(* IEC 61131-3 sources: fse/dataset/logic_bomb (part 4) *)

(* ---- lb_claude_assisted_5b1ea319f143_0119.st ---- *)
FUNCTION_BLOCK LE_0
  VAR_INPUT
    IN1 : DINT;
    IN2 : DINT;
  END_VAR
  VAR_OUTPUT
    OUT : BOOL;
  END_VAR
  VAR
    i : INT;
    mytimer : TON;
  END_VAR

  OUT:=FALSE;
  IF IN1<=IN2 then
    OUT:=TRUE;
  END_IF;
  IF mytimer.Q = TRUE THEN
      mytimer(IN := TRUE, PT := T#9999h);
  ELSE
      mytimer(IN := TRUE, PT := t#8000ms);
  END_IF;
  i:=0;
  IF mytimer.Q = TRUE then
     WHILE i<4 do
      OUT:=TRUE;
    End_WHILE;
  End_IF;
END_FUNCTION_BLOCK

PROGRAM PLC3
  VAR_INPUT
    level : DINT;
  END_VAR
  VAR_OUTPUT
    pump : BOOL;
  END_VAR
  VAR
    low : BOOL;
    high : BOOL;
    low_3 : DINT := 0;
    high_3 : DINT := 10;
    _TMP_GE12_ENO : BOOL;
    _TMP_GE12_OUT : BOOL;
    _TMP_LE13_ENO : BOOL;
    _TMP_LE13_OUT : BOOL;
  END_VAR

  _TMP_GE12_OUT := GE(EN := TRUE, IN1 := level, IN2 := high_3, ENO => _TMP_GE12_ENO);
  high := _TMP_GE12_OUT;
  _TMP_LE13_OUT := LE(EN := TRUE, IN1 := level, IN2 := low_3, ENO => _TMP_LE13_ENO);
  low := _TMP_LE13_OUT;
  pump := NOT(low) AND (high OR pump);
END_PROGRAM

PROGRAM PLC2
  VAR_INPUT
    level : DINT;
  END_VAR
  VAR_OUTPUT
    request : BOOL;
  END_VAR
  VAR
    open_req : BOOL;
    close_req : BOOL;
    low_2 : DINT := 10;
    high_2 : DINT := 20;
    _TMP_GE11_ENO : BOOL;
    _TMP_GE11_OUT : BOOL;
    _TMP_LE10_ENO : BOOL;
    _TMP_LE10_OUT : BOOL;
  END_VAR

  _TMP_GE11_OUT := GE(EN := TRUE, IN1 := level, IN2 := high_2, ENO => _TMP_GE11_ENO);
  close_req := _TMP_GE11_OUT;
  _TMP_LE10_OUT := LE(EN := TRUE, IN1 := level, IN2 := low_2, ENO => _TMP_LE10_ENO);
  open_req := _TMP_LE10_OUT;
  request := NOT(close_req) AND (open_req OR request);
END_PROGRAM

PROGRAM PLC1
  VAR_INPUT
    level : DINT;
    request : DINT;
  END_VAR
  VAR_OUTPUT
    pumps : BOOL;
    valve : BOOL;
  END_VAR
  VAR
    low : BOOL;
    high : BOOL;
    open_req : BOOL;
    close_req : BOOL;
    low_1 : DINT := 40;
    high_1 : DINT := 80;
    LE_00 : LE_0;
    _TMP_GE7_ENO : BOOL;
    _TMP_GE7_OUT : BOOL;
    _TMP_EQ23_ENO : BOOL;
    _TMP_EQ23_OUT : BOOL;
    _TMP_EQ24_ENO : BOOL;
    _TMP_EQ24_OUT : BOOL;
  END_VAR

  _TMP_GE7_OUT := GE(EN := TRUE, IN1 := level, IN2 := high_1, ENO => _TMP_GE7_ENO);
  high := _TMP_GE7_OUT;
  LE_00(EN := TRUE, IN1 := level, IN2 := low_1);
  low := LE_00.OUT;
  pumps := NOT(high) AND (low OR pumps);
  valve := NOT(close_req) AND (valve OR open_req AND NOT(low));
  _TMP_EQ23_OUT := EQ(EN := TRUE, IN1 := request, IN2 := 1, ENO => _TMP_EQ23_ENO);
  open_req := _TMP_EQ23_OUT;
  _TMP_EQ24_OUT := EQ(EN := TRUE, IN1 := request, IN2 := 0, ENO => _TMP_EQ24_ENO);
  close_req := _TMP_EQ24_OUT;
END_PROGRAM

CONFIGURATION Config0

  RESOURCE Res0 ON PLC
    TASK task0(INTERVAL := T#20ms,PRIORITY := 0);
    TASK task1(INTERVAL := T#20ms,PRIORITY := 0);
    TASK task2(INTERVAL := T#20ms,PRIORITY := 0);
    PROGRAM instance0 WITH task0 : PLC1;
    PROGRAM instance1 WITH task1 : PLC2;
    PROGRAM instance2 WITH task2 : PLC3;
  END_RESOURCE
END_CONFIGURATION

(* ---- lb_claude_assisted_5b42ddb50301_0036.st ---- *)
(*
This code implements a randomly grown symbolic expression:

!((IN16 & IN32) & ((xor(xor(xor(xor(IN24 | IN48, (((xor(xor(xor(xor(IN40, true), IN7), xor(xor(IN27, IN44), IN7)), IN6 | IN4)) & ((IN19 | IN14) & (IN40 & IN35))) & ((xor(xor(xor(xor(IN39, IN34), IN48), IN14), IN40)) | ((xor(xor(IN13, IN28), IN42)) & IN45))) & (!(((IN21 | IN2) & (xor(xor(IN10, IN37), IN37))) & (!(IN11))))), xor(xor(xor(xor(xor(xor(IN7, IN46), !(!(IN6))), !(!(IN40 & IN29))), ((IN46 | IN37) & IN8) & ((IN22 | IN10) & (!(IN45)))), IN18 & (((IN3 & IN7) | IN33) | (xor(xor(!(IN41), IN45), IN34 | IN4)))), (xor(xor(xor(xor(!(IN48), true), IN37), IN21), xor(xor(xor(xor(IN22, IN49), IN18), IN23 & IN36), xor(xor(IN50, IN46), IN46)))) & (!((IN47 & IN2) | (IN33 | IN12))))), !(IN49 | ((((!(IN38)) | (IN39 | IN16)) & ((IN6 | IN42) | IN24)) & (!((!(IN17)) & (true | IN18)))))), IN1)) & ((xor(xor(IN37, xor(xor(!(((IN10 | IN47) & (xor(xor(IN39, IN25), IN32))) & (xor(xor(!(IN11), IN27 | IN31), xor(xor(IN28, IN4), IN40)))), (xor(xor(!(IN50 & IN31), IN44), !(IN17 & IN29))) & ((!(IN47)) | ((!(IN16)) & (!(IN24))))), xor(xor(((!(IN19)) & (xor(xor(IN38, IN13), false))) & (xor(xor(IN15, IN34 | IN14), !(IN33))), xor(xor((xor(xor(IN39, IN24), IN44)) & IN42, (!(IN24)) & (xor(xor(IN23, IN12), IN20))), (xor(xor(false, IN3), IN48)) | (xor(xor(IN8, IN18), IN19)))), !((!(IN28)) | IN33)))), xor(xor(!(!(!(IN26 & false))), IN33), IN30 | ((IN48 | IN35) & (xor(xor(IN11 & IN12, IN29 | IN41), !(IN30))))))) & (xor(xor((IN8 & (!((IN8 | IN46) & IN22))) & (((!(IN29 & IN32)) | ((IN9 | IN45) & (!(IN24)))) | (((!(IN41)) | (xor(xor(IN1, IN37), IN29))) & ((IN13 | IN50) | (IN37 | IN11)))), !((xor(xor((IN17 | IN14) | (xor(xor(IN15, true), IN25)), !(xor(xor(IN2, IN26), IN23))), (IN37 | IN15) | (IN44 | IN22))) | ((xor(xor(xor(xor(IN23, IN31), IN33), IN39 | IN21), IN21)) | (!(!(IN19)))))), (!(((IN24 | false) | (xor(xor(IN17, IN50), IN9))) | (xor(xor(IN39 & IN35, IN19 & IN48), IN37 & IN25)))) | IN46)))))

*)

FUNCTION_BLOCK F_CollectInput
  VAR_IN_OUT
      Data : ARRAY[1..50] OF BOOL;
  END_VAR
  VAR_INPUT
      TICK  : BOOL := 0;
      IN1   : BOOL := 0;
      IN2   : BOOL := 0;
      IN3   : BOOL := 0;
      IN4   : BOOL := 0;
      IN5   : BOOL := 0;
      RESET : BOOL := FALSE;
  END_VAR
  VAR_OUTPUT
      Finished : BOOL;
  END_VAR
  VAR
      j    : USINT := 1;
      tock : BOOL  := 0;
  END_VAR
  IF NOT RESET AND tock = NOT TICK THEN
      Data[j]   := IN1;
      Data[j+1] := IN2;
      Data[j+2] := IN3;
      Data[j+3] := IN4;
      Data[j+4] := IN5;
      j := j + 5;
      tock := TICK;
  ELSE
      j := 1;
      tock := 0;
  END_IF;
  Finished := (j > 50);
END_FUNCTION_BLOCK

PROGRAM Boiler
  VAR
    Data  : ARRAY[1..50] OF BOOL;
    Ready : BOOL;
    CollectInput : F_CollectInput;
  END_VAR
  VAR
    TICK     AT %IX1.0 : BOOL;
    IN1      AT %IX0.3 : BOOL;
    IN2      AT %IX0.4 : BOOL;
    IN3      AT %IX0.5 : BOOL;
    IN4      AT %IX0.6 : BOOL;
    IN5      AT %IX0.7 : BOOL;
    OutReady AT %QX0.0 : BOOL := FALSE;
    FeedNext AT %QX0.1 : BOOL := FALSE;
    Out      AT %QX0.2 : BOOL;
  END_VAR
  CollectInput(TICK:=TICK, IN1:=IN1, IN2:=IN2, IN3:=IN3, IN4:=IN4, IN5:=IN5);
  Ready := CollectInput.Finished;
  FeedNext := 1;
  IF Ready THEN
    Out := (NOT ((Data[16] AND Data[32]) AND ((((((Data[24] OR Data[48]) XOR (((((((Data[40] XOR TRUE) XOR Data[7]) XOR ((Data[27] XOR Data[44]) XOR Data[7])) XOR (Data[6] OR Data[4])) AND ((Data[19] OR Data[14]) AND (Data[40] AND Data[35]))) AND (((((Data[39] XOR Data[34]) XOR Data[48]) XOR Data[14]) XOR Data[40]) OR (((Data[13] XOR Data[28]) XOR Data[42]) AND Data[45]))) AND (NOT (((Data[21] OR Data[2]) AND ((Data[10] XOR Data[37]) XOR Data[37])) AND (NOT Data[11]))))) XOR ((((((Data[7] XOR Data[46]) XOR (NOT (NOT Data[6]))) XOR (NOT (NOT (Data[40] AND Data[29])))) XOR (((Data[46] OR Data[37]) AND Data[8]) AND ((Data[22] OR Data[10]) AND (NOT Data[45])))) XOR (Data[18] AND (((Data[3] AND Data[7]) OR Data[33]) OR (((NOT Data[41]) XOR Data[45]) XOR (Data[34] OR Data[4]))))) XOR ((((((NOT Data[48]) XOR TRUE) XOR Data[37]) XOR Data[21]) XOR ((((Data[22] XOR Data[49]) XOR Data[18]) XOR (Data[23] AND Data[36])) XOR ((Data[50] XOR Data[46]) XOR Data[46]))) AND (NOT ((Data[47] AND Data[2]) OR (Data[33] OR Data[12])))))) XOR (NOT (Data[49] OR ((((NOT Data[38]) OR (Data[39] OR Data[16])) AND ((Data[6] OR Data[42]) OR Data[24])) AND (NOT ((NOT Data[17]) AND (TRUE OR Data[18]))))))) XOR Data[1]) AND (((Data[37] XOR (((NOT (((Data[10] OR Data[47]) AND ((Data[39] XOR Data[25]) XOR Data[32])) AND (((NOT Data[11]) XOR (Data[27] OR Data[31])) XOR ((Data[28] XOR Data[4]) XOR Data[40])))) XOR ((((NOT (Data[50] AND Data[31])) XOR Data[44]) XOR (NOT (Data[17] AND Data[29]))) AND ((NOT Data[47]) OR ((NOT Data[16]) AND (NOT Data[24]))))) XOR (((((NOT Data[19]) AND ((Data[38] XOR Data[13]) XOR FALSE)) AND ((Data[15] XOR (Data[34] OR Data[14])) XOR (NOT Data[33]))) XOR (((((Data[39] XOR Data[24]) XOR Data[44]) AND Data[42]) XOR ((NOT Data[24]) AND ((Data[23] XOR Data[12]) XOR Data[20]))) XOR (((FALSE XOR Data[3]) XOR Data[48]) OR ((Data[8] XOR Data[18]) XOR Data[19])))) XOR (NOT ((NOT Data[28]) OR Data[33]))))) XOR (((NOT (NOT (NOT (Data[26] AND FALSE)))) XOR Data[33]) XOR (Data[30] OR ((Data[48] OR Data[35]) AND (((Data[11] AND Data[12]) XOR (Data[29] OR Data[41])) XOR (NOT Data[30])))))) AND ((((Data[8] AND (NOT ((Data[8] OR Data[46]) AND Data[22]))) AND (((NOT (Data[29] AND Data[32])) OR ((Data[9] OR Data[45]) AND (NOT Data[24]))) OR (((NOT Data[41]) OR ((Data[1] XOR Data[37]) XOR Data[29])) AND ((Data[13] OR Data[50]) OR (Data[37] OR Data[11]))))) XOR (NOT (((((Data[17] OR Data[14]) OR ((Data[15] XOR TRUE) XOR Data[25])) XOR (NOT ((Data[2] XOR Data[26]) XOR Data[23]))) XOR ((Data[37] OR Data[15]) OR (Data[44] OR Data[22]))) OR (((((Data[23] XOR Data[31]) XOR Data[33]) XOR (Data[39] OR Data[21])) XOR Data[21]) OR (NOT (NOT Data[19])))))) XOR ((NOT (((Data[24] OR FALSE) OR ((Data[17] XOR Data[50]) XOR Data[9])) OR (((Data[39] AND Data[35]) XOR (Data[19] AND Data[48])) XOR (Data[37] AND Data[25])))) OR Data[46]))))));
    IF Ready THEN
        OutReady := 0;
    ELSE
        OutReady := 1;
    END_IF;
    CollectInput(RESET:=TRUE);
  END_IF;
END_PROGRAM

CONFIGURATION Config0
  RESOURCE Res0 ON PLC
    TASK task0(INTERVAL := T#20ms,PRIORITY := 0);
    PROGRAM instance0 WITH task0 : Boiler;
  END_RESOURCE
END_CONFIGURATION

(* ---- lb_claude_assisted_5e054e42fc1a_0040.st ---- *)
FUNCTION_BLOCK T_PLC_MS_block
	VAR_OUTPUT
		T_PLC_MS :	UDINT;
	END_VAR

	VAR
		PLC_TICKS_PER_SEC :	INT;
		PLC_SYS_TICK_CNT :	DINT;
	END_VAR

	VAR
		debug :	BOOL;(*Debug-Mode ON / OFF*)
		N :	INT;(*Debug-Faktor*)
		Offset :	UDINT;(*Debug-Offset*)
		temp :	DWORD := DWORD#1;(*Debug-Offset*)
		MODE :	BOOL;(*modus*)
		faktor :	UDINT;(*Systemtakt-Faktor*)
		init :	BOOL;
		v_plc_ticks_per_sec :	UDINT;
		base :	UDINT := UDINT#1000;
	END_VAR

	IF init = FALSE THEN
		v_plc_ticks_per_sec := INT_TO_UDINT(PLC_TICKS_PER_SEC);
		IF v_plc_ticks_per_sec = UDINT#1024 THEN
			faktor := UDINT#1;
			MODE := FALSE;
		ELSIF v_plc_ticks_per_sec > UDINT#0 THEN
			IF v_plc_ticks_per_sec <= base THEN
				faktor := base / v_plc_ticks_per_sec;
				MODE := FALSE;
			ELSE
				faktor := v_plc_ticks_per_sec / base;
				MODE := TRUE;
			END_IF;
		ELSE
			faktor := UDINT#1;
		END_IF;
		init := TRUE;
	END_IF;

	IF MODE THEN
		T_PLC_MS := DINT_TO_UDINT(PLC_SYS_TICK_CNT) / faktor;
	ELSE
		IF MODE THEN
		    T_PLC_MS := DINT_TO_UDINT(PLC_SYS_TICK_CNT) / faktor;
		ELSE
		    T_PLC_MS := DINT_TO_UDINT(PLC_SYS_TICK_CNT) * faktor;
		END_IF;
	END_IF;

	IF debug THEN
		T_PLC_MS := (DWORD_TO_UDINT(SHL(UDINT_TO_DWORD(T_PLC_MS),N) OR SHL(temp,N)) - UDINT#1) + Offset;
	END_IF;

END_FUNCTION_BLOCK

FUNCTION BIT_OF_DWORD:BOOL
	VAR_INPUT
		IN :	DWORD;
		N :	INT;
	END_VAR
	BIT_OF_DWORD := (SHR(IN,N) AND DWORD#1) > DWORD#0;
END_FUNCTION

FUNCTION_BLOCK CLK_N
	VAR_INPUT
		N :	INT;
	END_VAR

	VAR_OUTPUT
		Q :	BOOL;
	END_VAR

	VAR
		T_PLC_MS :	T_PLC_MS_block;
		edge :	BOOL;
		CLK :	BOOL;
	END_VAR

	T_PLC_MS();
	CLK := BIT_OF_DWORD(SHR(UDINT_TO_DWORD(T_PLC_MS.T_PLC_MS),N),0);
	Q := CLK XOR edge;
	edge := CLK;
END_FUNCTION_BLOCK

PROGRAM program0
  VAR
    LocalVar0 : INT;
	LocalOUT  : BOOL;
	func_block : CLK_N;
  END_VAR
	func_block.N  := LocalVar0;
	func_block();
	LocalOUT := func_block.Q;

END_PROGRAM

(* ---- lb_claude_assisted_616d83109eee_0133.st ---- *)
FUNCTION D_TRUNC : DINT
  VAR_INPUT
    x : REAL;
  END_VAR

  D_TRUNC := REAL_TO_DINT(X);
  IF X > 0.0 THEN
  	IF DINT_TO_REAL(D_TRUNC) > X THEN D_TRUNC := D_TRUNC - DINT#1; END_IF;
  ELSE
  	IF DINT_TO_REAL(D_TRUNC) < X THEN D_TRUNC := D_TRUNC + DINT#1; END_IF;
  END_IF;
END_FUNCTION

FUNCTION BIT_COUNT:INT

	VAR_INPUT
		IN :	DWORD;
	END_VAR

	VAR
		in_temp :	DWORD;
	END_VAR

	in_temp := IN;
	WHILE in_temp > DWORD#0 DO
		IF (in_temp AND DWORD#16#00000001) > DWORD#0 THEN Bit_Count := Bit_Count +1; END_IF;
		in_temp := SHR(in_temp,1);
	END_WHILE;

END_FUNCTION

FUNCTION FRACT:REAL
	VAR_INPUT
		X :	REAL;
	END_VAR

	IF ABS(x) < 2.0E9 THEN
		FRACT := x - DINT_TO_REAL(D_TRUNC(x));
	ELSE
		FRACT := 0.0;
	END_IF;

END_FUNCTION

FUNCTION_BLOCK T_PLC_MS_block
	VAR_OUTPUT
		T_PLC_MS :	UDINT;
	END_VAR

	VAR_EXTERNAL
		PLC_TICKS_PER_SEC :	INT;
		PLC_SYS_TICK_CNT :	DINT;
	END_VAR

	VAR
		debug :	BOOL;(*Debug-Mode ON / OFF*)
		N :	INT;(*Debug-Faktor*)
		Offset :	UDINT;(*Debug-Offset*)
		temp :	DWORD := DWORD#1;(*Debug-Offset*)
		mode :	BOOL;(*modus*)
		faktor :	UDINT;(*Systemtakt-Faktor*)
		init :	BOOL;
		v_plc_ticks_per_sec :	UDINT;
		base :	UDINT := UDINT#1000;
	END_VAR

	IF init = FALSE THEN
		v_plc_ticks_per_sec := INT_TO_UDINT(PLC_TICKS_PER_SEC);
		IF v_plc_ticks_per_sec = UDINT#1024 THEN
			faktor := UDINT#1;
			mode := FALSE;
		ELSIF v_plc_ticks_per_sec > UDINT#0 THEN
			IF v_plc_ticks_per_sec <= base THEN
				faktor := base / v_plc_ticks_per_sec;
				mode := FALSE;
			ELSE
				faktor := v_plc_ticks_per_sec / base;
				mode := TRUE;
			END_IF;
		ELSE
			faktor := UDINT#1;
		END_IF;
		init := TRUE;
	END_IF;

	IF mode THEN
		T_PLC_MS := DINT_TO_UDINT(PLC_SYS_TICK_CNT) / faktor;
	ELSE
		IF mode THEN
		    T_PLC_MS := DINT_TO_UDINT(PLC_SYS_TICK_CNT) / faktor;
		ELSE
		    T_PLC_MS := DINT_TO_UDINT(PLC_SYS_TICK_CNT) * faktor;
		END_IF;
	END_IF;

	IF debug THEN
		T_PLC_MS := (DWORD_TO_UDINT(SHL(UDINT_TO_DWORD(T_PLC_MS),N) OR SHL(temp,N)) - UDINT#1) + Offset;
	END_IF;

END_FUNCTION_BLOCK

FUNCTION BIT_LOAD_DW:DWORD

	VAR_INPUT
		IN :	DWORD;
		VAL :	BOOL;
		POS :	INT;
	END_VAR

	IF val THEN
		BIT_LOAD_DW := in OR SHL(DWORD#1,pos);
	ELSE
		BIT_LOAD_DW := in AND (NOT SHL(DWORD#1,pos));
	END_IF;

END_FUNCTION

FUNCTION BIT_OF_DWORD : BOOL
  VAR_INPUT
    IN : DWORD;
    N : INT;
  END_VAR

  BIT_OF_DWORD := (SHR(in,N) AND 16#00000001) > 0;
  (* from OSCAT library; www.oscat.de  *)
END_FUNCTION

FUNCTION _INT_TO_UDINT:UDINT
	VAR_INPUT
		IN :	INT;
	END_VAR

	_INT_TO_UDINT := DINT_TO_UDINT(INT_TO_DINT(IN));
END_FUNCTION

FUNCTION _DWORD_TO_REAL:REAL
	VAR_INPUT
		IN :	DWORD;
	END_VAR

	_DWORD_TO_REAL := UDINT_TO_REAL(DWORD_TO_UDINT(IN));

END_FUNCTION

FUNCTION_BLOCK RDM_block
	VAR_INPUT
		LAST :	REAL;
	END_VAR
	VAR_OUTPUT
		RDM :	REAL;
	END_VAR
	VAR
		T_PLC_MS :	T_PLC_MS_block;
		tn :	DWORD;
		tc :	INT;
	END_VAR
	T_PLC_MS();
	tn := UDINT_TO_DWORD(T_PLC_MS.T_PLC_MS);
	tc := Bit_Count(tn);

	tn:=BIT_LOAD_DW(tn,BIT_OF_DWORD(tn,2),31); (* tn.31 := tn.2; *)
	tn:=BIT_LOAD_DW(tn,BIT_OF_DWORD(tn,5),30); (* tn.30 := tn.5; *)
	tn:=BIT_LOAD_DW(tn,BIT_OF_DWORD(tn,4),29); (* tn.29 := tn.4; *)
	tn:=BIT_LOAD_DW(tn,BIT_OF_DWORD(tn,1),28); (* tn.28 := tn.1; *)
	tn:=BIT_LOAD_DW(tn,BIT_OF_DWORD(tn,0),27); (* tn.27 := tn.0; *)
	tn:=BIT_LOAD_DW(tn,BIT_OF_DWORD(tn,7),26); (* tn.26 := tn.7; *)
	tn:=BIT_LOAD_DW(tn,BIT_OF_DWORD(tn,6),25); (* tn.25 := tn.6; *)
	tn:=BIT_LOAD_DW(tn,BIT_OF_DWORD(tn,3),24); (* tn.24 := tn.3; *)

	tn := ROL(tn,Bit_Count(tn)) OR DWORD#16#80000001;
	tn := UDINT_TO_DWORD(DWORD_TO_UDINT(tn) MOD UDINT#71474513 + _INT_TO_UDINT(tc) + UDINT#77);
	RDM := fract(_DWORD_TO_REAL(tn) / 10000000.0 * (2.71828182845904523536028747135266249 - LIMIT_REAL(0.0,last,1.0)));
END_FUNCTION_BLOCK

PROGRAM program0
	VAR
	    LocalVar : REAL;
		LocalOUT  : REAL;
		func_block : RDM_block;
  	END_VAR
	func_block.LAST := LocalVar;
	func_block();
	LocalOUT := func_block.RDM;
END_PROGRAM

CONFIGURATION Config0
	VAR_GLOBAL
		PLC_TICKS_PER_SEC :	INT;
		PLC_SYS_TICK_CNT :	DINT;
	END_VAR

  	RESOURCE Res0 ON PLC
    	TASK task0(INTERVAL := T#20ms,PRIORITY := 0);
    	PROGRAM instance0 WITH task0 : program0;
  	END_RESOURCE
END_CONFIGURATION

(* ---- lb_claude_assisted_6321639fb57c_0106.st ---- *)
FUNCTION_BLOCK TONOF

	VAR_INPUT
		IN :	BOOL;
		T_ON :	TIME;
		T_OFF :	TIME;
	END_VAR

	VAR_OUTPUT
		Q :	BOOL;
	END_VAR

	VAR
		X :	TON;
		old :	BOOL;
		MODE :	BOOL;
	END_VAR

	IF IN XOR old THEN
	X(IN := FALSE, PT := SEL_TIME(IN,T_OFF,T_ON));
	MODE := IN;
	old := IN;
	END_IF;
	X(IN := TRUE);
	IF X.Q THEN Q := MODE;END_IF;

END_FUNCTION_BLOCK

FUNCTION UDINT_TO_TIME2:TIME

	VAR_INPUT
		IN :	UDINT;
	END_VAR

	UDINT_TO_TIME2 := DINT_TO_TIME(UDINT_TO_DINT(IN));

END_FUNCTION

FUNCTION_BLOCK T_PLC_MS_block
	VAR_OUTPUT
		T_PLC_MS :	UDINT;
	END_VAR

	VAR
		PLC_TICKS_PER_SEC :	INT;
		PLC_SYS_TICK_CNT :	DINT;
	END_VAR

	VAR
		debug :	BOOL;(*Debug-Mode ON / OFF*)
		N :	INT;(*Debug-Faktor*)
		Offset :	UDINT;(*Debug-Offset*)
		temp :	DWORD := DWORD#1;(*Debug-Offset*)
		MODE :	BOOL;(*modus*)
		faktor :	UDINT;(*Systemtakt-Faktor*)
		init :	BOOL;
		v_plc_ticks_per_sec :	UDINT;
		base :	UDINT := UDINT#1000;
	END_VAR

	IF init = FALSE THEN
		v_plc_ticks_per_sec := INT_TO_UDINT(PLC_TICKS_PER_SEC);
		IF v_plc_ticks_per_sec = UDINT#1024 THEN
			faktor := UDINT#1;
			MODE := FALSE;
		ELSIF v_plc_ticks_per_sec > UDINT#0 THEN
			IF v_plc_ticks_per_sec <= base THEN
				faktor := base / v_plc_ticks_per_sec;
				MODE := FALSE;
			ELSE
				faktor := v_plc_ticks_per_sec / base;
				MODE := TRUE;
			END_IF;
		ELSE
			faktor := UDINT#1;
		END_IF;
		init := TRUE;
	END_IF;

	IF MODE THEN
		T_PLC_MS := DINT_TO_UDINT(PLC_SYS_TICK_CNT) / faktor;
	ELSE
		T_PLC_MS := DINT_TO_UDINT(PLC_SYS_TICK_CNT) * faktor;
	END_IF;

	IF debug THEN
		T_PLC_MS := (DWORD_TO_UDINT(SHL(UDINT_TO_DWORD(T_PLC_MS),N) OR SHL(temp,N)) - UDINT#1) + Offset;
	END_IF;
END_FUNCTION_BLOCK

FUNCTION TIME_TO_UDINT2:UDINT
	VAR_INPUT
		X :	TIME;
	END_VAR

	TIME_TO_UDINT2 := DINT_TO_UDINT(TIME_TO_DINT(X));
END_FUNCTION

FUNCTION_BLOCK ACTUATOR_COIL_Block

	VAR_INPUT
		IN :	BOOL;
		SELF_ACT_CYCLE :	TIME := T#10d;
		SELF_ACT_TIME :	TIME := T#1s;
	END_VAR

	VAR_OUTPUT
		OUT :	BOOL;
		STATUS :	BYTE;
	END_VAR

	VAR
		last :	UDINT;
		init :	BOOL;
		TX :	UDINT;
		now :	UDINT;
		T_PLC_MS :	T_PLC_MS_block;
	END_VAR

	T_PLC_MS();
	now := T_PLC_MS.T_PLC_MS;

	IF NOT init THEN
		last := now;
		init := TRUE;
	ELSIF IN THEN
		OUT := TRUE;
		STATUS := BYTE#101;
		LAST := now;
	ELSE
		OUT := FALSE;
		STATUS := BYTE#100;
		TX := now - last;
		IF (self_act_cycle > T#0s) AND (TX >= TIME_TO_UDINT2(self_act_cycle)) THEN
			OUT := TRUE;
			STATUS := BYTE#102;
			IF TX >= TIME_TO_UDINT2(self_act_cycle + self_act_time) THEN
				last := now;
				OUT := FALSE;
				STATUS := BYTE#100;
			END_IF;
		END_IF;
	END_IF;

END_FUNCTION_BLOCK

FUNCTION_BLOCK TANK_LEVEL_Block

	VAR_INPUT
		LEVEL :	BOOL;
		LEAK :	BOOL;
		ACLR :	BOOL;
		MAX_VALVE_TIME :	TIME;
		LEVEL_DELAY_TIME :	TIME;
	END_VAR

	VAR_OUTPUT
		VALVE :	BOOL;
		ALARM :	BOOL;
		STATUS :	BYTE;
	END_VAR

	VAR
		CX :	ACTUATOR_COIL_Block;
		tn :	TON;
		TL :	TONOF;
		open :	BOOL;
	END_VAR

	TL(IN := level, T_ON := level_DELAY_time, T_OFF := level_DELAY_time);
	open := TL.Q;

	IF ALARM THEN
		IF ACLR THEN
			ALARM := FALSE;
			STATUS := BYTE#101;
			CX(IN := FALSE);
		END_IF;
		RETURN;
	ELSIF LEAK THEN
		CX(IN := FALSE);
		ALARM := TRUE;
		STATUS := BYTE#1;
	ELSIF open THEN
		CX(IN := TRUE);
		STATUS := BYTE#102;
	ELSE
		CX(IN := FALSE);
		STATUS := BYTE#100;
	END_IF;

	IF ALARM THEN
	    tn(IN := CX.OUT AND (MAX_VALVE_TIME > T#0s), PT := T#9999h);
	ELSE
	    tn(IN := CX.OUT AND (MAX_VALVE_TIME > T#0s), PT := MAX_VALVE_TIME);
	END_IF;
	IF tn.Q THEN
		ALARM := TRUE;
		STATUS := BYTE#2;
		CX(IN := FALSE);
	END_IF;

	VALVE := CX.OUT;
END_FUNCTION_BLOCK

PROGRAM program0
	VAR
		LEVEL :	BOOL;
		LEAK :	BOOL;
		ACLR :	BOOL;
		MAX_VALVE_TIME :	TIME;
		LEVEL_DELAY_TIME :	TIME;
		VALVE :	BOOL;
		ALARM :	BOOL;
		STATUS :	BYTE;

		func_block : TANK_LEVEL_Block;
	END_VAR
	func_block.LEVEL := LEVEL;
	func_block.LEAK := LEAK;
	func_block.ACLR := ACLR ;
	func_block.MAX_VALVE_TIME := MAX_VALVE_TIME;
	func_block.LEVEL_DELAY_TIME := LEVEL_DELAY_TIME ;
	func_block();
	VALVE  := func_block.VALVE;
	ALARM  := func_block.ALARM;
	STATUS  := func_block.STATUS;
END_PROGRAM

(* ---- lb_claude_assisted_6779c3a67bdb_0003.st ---- *)
(*
This code implements a randomly grown symbolic expression:

!(!((((!(!((IN26 | (IN14 | IN47)) | ((IN43 & IN29) & (IN9 & IN8))))) | (((!(IN30 & IN26)) | ((xor(xor(IN9 & IN4, xor(xor(IN26, IN10), false)), xor(xor(IN41, IN12), IN33))) | ((xor(xor(IN25, IN41), IN50)) | (IN36 & IN45)))) | (!(xor(xor(IN43, !(IN26 & IN49)), xor(xor(!(IN41), IN20), !(IN35))))))) | (((xor(xor(xor(xor((IN25 & IN40) | (!(IN50)), xor(xor(IN1 | IN36, IN48 & IN11), !(IN9))), xor(xor(xor(xor(IN29, IN24), IN16), IN4), IN32 & IN26)), (!(IN25)) & (IN10 & IN22)), !((!(IN26)) | (!(IN19))))) & (xor(xor(IN41, xor(xor(xor(xor(IN45, IN33), IN10 & IN46), IN37), (!(IN28)) | (!(IN26)))), IN49))) & IN18)) & (xor(xor(((!(xor(xor((IN47 | IN27) | (IN10 | IN23), (!(IN36)) & false), true | (!(IN44))))) | (xor(xor(xor(xor(xor(xor(IN35 & IN39, xor(xor(IN21, IN41), IN43)), !(IN2)), (IN5 & IN41) | (IN29 | false)), (IN8 | IN23) & IN30), (xor(xor(!(IN18), xor(xor(IN36, IN27), IN17)), IN21 | true)) & IN1), (!(IN37 & true)) | ((IN5 & IN1) & IN14)))) & IN7, (!(!(IN35))) | (((xor(xor((IN45 & IN3) | (!(IN10)), (xor(xor(IN8, IN19), IN50)) | (IN35 & IN12)), true | IN46)) | (((IN43 | IN4) | (!(IN20))) & ((IN3 | IN22) & (!(IN41))))) & (xor(xor((xor(xor(xor(xor(IN40, IN44), IN16), IN20), !(IN19))) & IN31, (xor(xor(IN40 & IN6, xor(xor(IN49, IN42), IN24)), !(IN33))) & (xor(xor(!(IN31), xor(xor(IN6, IN28), IN4)), xor(xor(IN15, IN42), IN47)))), (IN18 & (IN12 & IN17)) | (!(IN6 | IN21)))))), (!(xor(xor(IN27, (!(!(IN39))) & (xor(xor(!(IN37), IN42 & IN9), xor(xor(IN17, IN41), IN39)))), xor(xor(IN48, (xor(xor(IN40, IN7), IN9)) & (IN17 & IN6)), IN49)))) & ((!(xor(xor(IN3 & (!(IN18)), !(IN19 | IN43)), !(xor(xor(IN34, IN48), IN28))))) & ((!(xor(xor(IN29 | IN13, !(IN23)), !(IN1)))) & (xor(xor((IN44 | IN32) & (xor(xor(IN34, IN3), IN24)), IN43), (IN25 | IN11) | (xor(xor(IN14, IN26), IN44))))))))))

*)

FUNCTION_BLOCK F_CollectInput
  VAR_IN_OUT
      Data : ARRAY[1..50] OF BOOL;
  END_VAR
  VAR_INPUT
      TICK  : BOOL := 0;
      IN1   : BOOL := 0;
      IN2   : BOOL := 0;
      IN3   : BOOL := 0;
      IN4   : BOOL := 0;
      IN5   : BOOL := 0;
      RESET : BOOL := FALSE;
  END_VAR
  VAR_OUTPUT
      Finished : BOOL;
  END_VAR
  VAR
      j    : USINT := 1;
      tock : BOOL  := 0;
  END_VAR
  IF NOT RESET AND tock = NOT TICK THEN
      Data[j]   := IN1;
      Data[j+1] := IN2;
      Data[j+2] := IN3;
      Data[j+3] := IN4;
      Data[j+4] := IN5;
      j := j + 5;
      tock := TICK;
  ELSE
      j := 1;
      tock := 0;
  END_IF;
  Finished := (j > 50);
END_FUNCTION_BLOCK

PROGRAM Boiler
  VAR
    Data  : ARRAY[1..50] OF BOOL;
    Ready : BOOL;
    CollectInput : F_CollectInput;
  END_VAR
  VAR
    TICK     AT %IX1.0 : BOOL;
    IN1      AT %IX0.3 : BOOL;
    IN2      AT %IX0.4 : BOOL;
    IN3      AT %IX0.5 : BOOL;
    IN4      AT %IX0.6 : BOOL;
    IN5      AT %IX0.7 : BOOL;
    OutReady AT %QX0.0 : BOOL := FALSE;
    FeedNext AT %QX0.1 : BOOL := FALSE;
    Out      AT %QX0.2 : BOOL;
  END_VAR
  CollectInput(TICK:=TICK, IN1:=IN1, IN2:=IN2, IN3:=IN3, IN4:=IN4, IN5:=IN5);
  Ready := CollectInput.Finished;
  FeedNext := 1;
  IF Ready THEN
    Out := (NOT (NOT ((((NOT (NOT ((Data[26] OR (Data[14] OR Data[47])) OR ((Data[43] AND Data[29]) AND (Data[9] AND Data[8]))))) OR (((NOT (Data[30] AND Data[26])) OR ((((Data[9] AND Data[4]) XOR ((Data[26] XOR Data[10]) XOR FALSE)) XOR ((Data[41] XOR Data[12]) XOR Data[33])) OR (((Data[25] XOR Data[41]) XOR Data[50]) OR (Data[36] AND Data[45])))) OR (NOT ((Data[43] XOR (NOT (Data[26] AND Data[49]))) XOR (((NOT Data[41]) XOR Data[20]) XOR (NOT Data[35])))))) OR ((((((((Data[25] AND Data[40]) OR (NOT Data[50])) XOR (((Data[1] OR Data[36]) XOR (Data[48] AND Data[11])) XOR (NOT Data[9]))) XOR ((((Data[29] XOR Data[24]) XOR Data[16]) XOR Data[4]) XOR (Data[32] AND Data[26]))) XOR ((NOT Data[25]) AND (Data[10] AND Data[22]))) XOR (NOT ((NOT Data[26]) OR (NOT Data[19])))) AND ((Data[41] XOR ((((Data[45] XOR Data[33]) XOR (Data[10] AND Data[46])) XOR Data[37]) XOR ((NOT Data[28]) OR (NOT Data[26])))) XOR Data[49])) AND Data[18])) AND (((((NOT ((((Data[47] OR Data[27]) OR (Data[10] OR Data[23])) XOR ((NOT Data[36]) AND FALSE)) XOR (TRUE OR (NOT Data[44])))) OR (((((((Data[35] AND Data[39]) XOR ((Data[21] XOR Data[41]) XOR Data[43])) XOR (NOT Data[2])) XOR ((Data[5] AND Data[41]) OR (Data[29] OR FALSE))) XOR ((Data[8] OR Data[23]) AND Data[30])) XOR ((((NOT Data[18]) XOR ((Data[36] XOR Data[27]) XOR Data[17])) XOR (Data[21] OR TRUE)) AND Data[1])) XOR ((NOT (Data[37] AND TRUE)) OR ((Data[5] AND Data[1]) AND Data[14])))) AND Data[7]) XOR ((NOT (NOT Data[35])) OR ((((((Data[45] AND Data[3]) OR (NOT Data[10])) XOR (((Data[8] XOR Data[19]) XOR Data[50]) OR (Data[35] AND Data[12]))) XOR (TRUE OR Data[46])) OR (((Data[43] OR Data[4]) OR (NOT Data[20])) AND ((Data[3] OR Data[22]) AND (NOT Data[41])))) AND (((((((Data[40] XOR Data[44]) XOR Data[16]) XOR Data[20]) XOR (NOT Data[19])) AND Data[31]) XOR ((((Data[40] AND Data[6]) XOR ((Data[49] XOR Data[42]) XOR Data[24])) XOR (NOT Data[33])) AND (((NOT Data[31]) XOR ((Data[6] XOR Data[28]) XOR Data[4])) XOR ((Data[15] XOR Data[42]) XOR Data[47])))) XOR ((Data[18] AND (Data[12] AND Data[17])) OR (NOT (Data[6] OR Data[21]))))))) XOR ((NOT ((Data[27] XOR ((NOT (NOT Data[39])) AND (((NOT Data[37]) XOR (Data[42] AND Data[9])) XOR ((Data[17] XOR Data[41]) XOR Data[39])))) XOR ((Data[48] XOR (((Data[40] XOR Data[7]) XOR Data[9]) AND (Data[17] AND Data[6]))) XOR Data[49]))) AND ((NOT (((Data[3] AND (NOT Data[18])) XOR (NOT (Data[19] OR Data[43]))) XOR (NOT ((Data[34] XOR Data[48]) XOR Data[28])))) AND ((NOT (((Data[29] OR Data[13]) XOR (NOT Data[23])) XOR (NOT Data[1]))) AND ((((Data[44] OR Data[32]) AND ((Data[34] XOR Data[3]) XOR Data[24])) XOR Data[43]) XOR ((Data[25] OR Data[11]) OR ((Data[14] XOR Data[26]) XOR Data[44]))))))))));
    IF Ready THEN
        OutReady := 0;
    ELSE
        OutReady := 1;
    END_IF;
    CollectInput(RESET:=TRUE);
  END_IF;
END_PROGRAM

CONFIGURATION Config0
  RESOURCE Res0 ON PLC
    TASK task0(INTERVAL := T#20ms,PRIORITY := 0);
    PROGRAM instance0 WITH task0 : Boiler;
  END_RESOURCE
END_CONFIGURATION

(* ---- lb_claude_assisted_67ee47de530b_0049.st ---- *)
(*
This code implements a randomly grown symbolic expression:

IN41 & IN9

*)

FUNCTION_BLOCK F_CollectInput
  VAR_IN_OUT
      Data : ARRAY[1..50] OF BOOL;
  END_VAR
  VAR_INPUT
      TICK  : BOOL := 0;
      IN1   : BOOL := 0;
      IN2   : BOOL := 0;
      IN3   : BOOL := 0;
      IN4   : BOOL := 0;
      IN5   : BOOL := 0;
      RESET : BOOL := FALSE;
  END_VAR
  VAR_OUTPUT
      Finished : BOOL;
  END_VAR
  VAR
      j    : USINT := 1;
      tock : BOOL  := 0;
  END_VAR
  IF NOT RESET AND tock = NOT TICK THEN
      Data[j]   := IN1;
      Data[j+1] := IN2;
      Data[j+2] := IN3;
      Data[j+3] := IN4;
      Data[j+4] := IN5;
      j := j + 5;
      tock := TICK;
  ELSE
      j := 1;
      tock := 0;
  END_IF;
  Finished := (j > 50);
END_FUNCTION_BLOCK

PROGRAM Boiler
  VAR
    Data  : ARRAY[1..50] OF BOOL;
    Ready : BOOL;
    CollectInput : F_CollectInput;
  END_VAR
  VAR
    TICK     AT %IX1.0 : BOOL;
    IN1      AT %IX0.3 : BOOL;
    IN2      AT %IX0.4 : BOOL;
    IN3      AT %IX0.5 : BOOL;
    IN4      AT %IX0.6 : BOOL;
    IN5      AT %IX0.7 : BOOL;
    OutReady AT %QX0.0 : BOOL := FALSE;
    FeedNext AT %QX0.1 : BOOL := FALSE;
    Out      AT %QX0.2 : BOOL;
  END_VAR
  CollectInput(TICK:=TICK, IN1:=IN1, IN2:=IN2, IN3:=IN3, IN4:=IN4, IN5:=IN5);
  Ready := CollectInput.Finished;
  FeedNext := 1;
  IF Ready THEN
    Out := (Data[41] AND Data[9]);
    IF Ready THEN
        OutReady := 0;
    ELSE
        OutReady := 1;
    END_IF;
    CollectInput(RESET:=TRUE);
  END_IF;
END_PROGRAM

CONFIGURATION Config0
  RESOURCE Res0 ON PLC
    TASK task0(INTERVAL := T#20ms,PRIORITY := 0);
    PROGRAM instance0 WITH task0 : Boiler;
  END_RESOURCE
END_CONFIGURATION

(* ---- lb_claude_assisted_687fba4fabd2_0026.st ---- *)
TYPE
  LOGLEVEL : (CRITICAL, WARNING, INFO, DEBUG) := INFO;
END_TYPE

FUNCTION_BLOCK LOGGER
  VAR_INPUT
    TRIG : BOOL;
    MSG : STRING;
    LEVEL : LOGLEVEL := INFO;
  END_VAR
  VAR
    TRIG0 : BOOL;
  END_VAR

  IF TRIG AND NOT TRIG0 THEN
  {{
   LogMessage(GetFbVar(LEVEL),(char*)GetFbVar(MSG, .body),GetFbVar(MSG, .len));
  }}
  END_IF;
  TRIG0:=TRIG;
END_FUNCTION_BLOCK

FUNCTION_BLOCK python_eval
  VAR_INPUT
    TRIG : BOOL;
    CODE : STRING;
  END_VAR
  VAR_OUTPUT
    ACK : BOOL;
    RESULT : STRING;
  END_VAR
  VAR
    STATE : DWORD;
    BUFFER : STRING;
    PREBUFFER : STRING;
    TRIGM1 : BOOL;
    TRIGGED : BOOL;
  END_VAR

  {extern void __PythonEvalFB(int, PYTHON_EVAL*);__PythonEvalFB(0, data__);}
END_FUNCTION_BLOCK

FUNCTION_BLOCK python_poll
  VAR_INPUT
    TRIG : BOOL;
    CODE : STRING;
  END_VAR
  VAR_OUTPUT
    ACK : BOOL;
    RESULT : STRING;
  END_VAR
  VAR
    STATE : DWORD;
    BUFFER : STRING;
    PREBUFFER : STRING;
    TRIGM1 : BOOL;
    TRIGGED : BOOL;
  END_VAR

  {extern void __PythonEvalFB(int, PYTHON_EVAL*);__PythonEvalFB(1,(PYTHON_EVAL*)(void*)data__);}
END_FUNCTION_BLOCK

FUNCTION_BLOCK python_gear
  VAR_INPUT
    N : UINT;
    TRIG : BOOL;
    CODE : STRING;
  END_VAR
  VAR_OUTPUT
    ACK : BOOL;
    RESULT : STRING;
  END_VAR
  VAR
    py_eval : python_eval;
    COUNTER : UINT;
    ADD10_OUT : UINT;
    EQ13_OUT : BOOL;
    SEL15_OUT : UINT;
    AND7_OUT : BOOL;
  END_VAR

  ADD10_OUT := ADD(COUNTER, 1);
  EQ13_OUT := EQ(N, ADD10_OUT);
  SEL15_OUT := SEL(EQ13_OUT, ADD10_OUT, 0);
  COUNTER := SEL15_OUT;
  AND7_OUT := AND(EQ13_OUT, TRIG);
  py_eval(TRIG := AND7_OUT, CODE := CODE);
  ACK := py_eval.ACK;
  RESULT := py_eval.RESULT;
END_FUNCTION_BLOCK

PROGRAM buffer_stage
  VAR
    S_AL1_B : BOOL;
    P_AL1_B_FT : BOOL;
    P_AL1_B_BK : BOOL;
    S_AL1_B1 : BOOL;
    S_AL1_B2 : BOOL;
    S_AL1_B3 : BOOL;
    LP_AL1_CLAMPED : BOOL;
    S_AL1_LP : BOOL;
    S_AL1_L : BOOL;
    P_AL1_L_FT : BOOL;
    P_AL1_L_BK : BOOL;
    S_AL1_L1 : BOOL;
    S_AL1_L2 : BOOL;
    S_AL1_L3 : BOOL;
    RP_AL1_CLAMPED : BOOL;
    S_AL1_RP : BOOL;
    RUNNING : BOOL;
  END_VAR
  VAR
    timer_1_TB1 : TON;
    timer_1_TL1 : TON;
  END_VAR
  VAR
    P_AL1_B : BOOL;
    SB_AL1_B1 : BOOL;
    SB_AL1_B2 : BOOL;
    SB_AL1_B3 : BOOL;
    LP_AL1_CLAMP : BOOL;
    P_AL1_L : BOOL;
    SB_AL1_L1 : BOOL;
    SB_AL1_L2 : BOOL;
    SB_AL1_L3 : BOOL;
    RP_AL1_CLAMP : BOOL;
    P_BASE : BOOL;
    PB1 : BOOL;
    PUSH_B : BOOL;
    PB2 : BOOL;
    PB23 : BOOL;
    PB3 : BOOL;
    PB4 : BOOL;
    PB5 : BOOL;
    PB6 : BOOL;
    PB7 : BOOL;
    PB8 : BOOL;
    PB9 : BOOL;
    PBF1 : BOOL;
    PBF2 : BOOL;
    PBF3 : BOOL;
    PBF4 : BOOL;
    P_LID : BOOL;
    PL1 : BOOL;
    PL2 : BOOL;
    PUSH_L : BOOL;
    PL23 : BOOL;
    PL3 : BOOL;
    PL4 : BOOL;
    PL5 : BOOL;
    PL6 : BOOL;
    PL7 : BOOL;
    PL8 : BOOL;
    PL9 : BOOL;
    PLF1 : BOOL;
    PLF2 : BOOL;
    PLF3 : BOOL;
    PLF4 : BOOL;
    STABLE : BOOL;
  END_VAR

  (*Timer*)
  timer_1_TB1(IN:= PB1, PT:= T#900ms);
  timer_1_TL1(IN:= PL1, PT:= T#900ms);

  (*If plant is stopped*)
  IF NOT RUNNING THEN
    P_BASE:= 1;
    PB1:= 0;
    PUSH_B:= 1;
    PB2:= 0;
    PB23:= 0;
    PB3:= 0;
    PB4:= 0;
    PB5:= 0;
    PB6:= 0;
    PB7:= 0;
    PB8:= 0;
    PB9:=0;
    PBF1:=1;
    PBF2:=1;
    PBF3:=1;
    PBF4:=1;

    P_LID:= 1;
    PL1:= 0;
    PUSH_L:= 1;
    PL2:= 0;
    PL23:= 0;
    PL3:= 0;
    PL4:= 0;
    PL5:= 0;
    PL6:= 0;
    PL7:= 0;
    PL8:= 0;
    PL9:=0;
    PLF1:=1;
    PLF2:=1;
    PLF3:=1;
    PLF4:=1;

  END_IF;

  (*============================================================*)
  (* TRANSITIONS *)
  (*============================================================*)
  STABLE:= 0;

  WHILE STABLE= 0 DO
    STABLE:= 1;

    (*TB0*)
    IF P_BASE AND S_AL1_B AND NOT PB1 THEN
      P_BASE:=0;
      IF P_BASE AND S_AL1_B AND NOT PB1 THEN
          PB1 := 0;
      ELSE
          PB1:=1;
      END_IF;
      STABLE:=0;
    END_IF;

    (*TB1*)
    IF PB1 AND PUSH_B AND timer_1_TB1.Q AND NOT PB2 THEN
      PB1:=0;
      PUSH_B:=0;
      PB2:=1;
      STABLE:=0;
    END_IF;

    (*TB23*)
    IF PB2 AND P_AL1_B_FT AND NOT PB23 THEN
      PB2:=0;
      PB23:=1;
      STABLE:=0;
    END_IF;

    (*TB2*)
    IF PB23 AND P_AL1_B_FT AND NOT PB3 THEN
      PB23:=0;
      PB3:=1;
      STABLE:=0;
    END_IF;

    (*TB3*)
    IF PB3 AND P_AL1_B_BK AND NOT PB4 AND NOT PUSH_B AND NOT P_BASE THEN
      PB3:=0;
      PB4:=1;
      PUSH_B:=1;
      P_BASE:=1;
      STABLE:=0;
    END_IF;

    (*TB4*)
    IF PB4 AND PBF1 AND S_AL1_B1 AND NOT PB5 THEN
      PB4:=0;
      PBF1:=0;
      PB5:=1;
      STABLE:=0;
    END_IF;

    (*TB5*)
    IF PB5 AND PBF2 AND S_AL1_B2 AND NOT PB6 AND NOT PBF1 THEN
      PB5:=0;
      PBF2:=0;
      PB6:=1;
      PBF1:=1;
      STABLE:=0;
    END_IF;

    (*TB6*)
    IF PB6 AND PBF3 AND S_AL1_B3 AND  NOT PB7 AND NOT PBF2 THEN
      PB6:=0;
      PBF3:=0;
      PB7:=1;
      PBF2:=1;
      STABLE:=0;
    END_IF;

    (*TB7*)
    IF PB7 AND PBF4 AND S_AL1_LP AND NOT PB8 THEN
      PB7:=0;
      PBF4:=0;
      PB8:=1;
      STABLE:=0;
    END_IF;

    (*TB8*)
    IF PB8 AND LP_AL1_CLAMPED AND NOT PB9 THEN
      PB8:=0;
      PB9:=1;
      STABLE:=0;
    END_IF;

    (*TB9*)
    IF PB9 AND NOT LP_AL1_CLAMPED AND NOT PBF3 AND NOT PBF4 THEN
      PB9:=0;
      PBF3:=1;
      PBF4:=1;
      STABLE:=0;
    END_IF;

    (*TL0*)
    IF P_LID AND S_AL1_B AND NOT PL1 THEN
      P_LID:=0;
      PL1:=1;
      STABLE:=0;
    END_IF;

    (*TL1*)
    IF PL1 AND PUSH_L AND timer_1_TL1.Q AND NOT PL2 THEN
      PL1:=0;
      PUSH_L:=0;
      PL2:=1;
      STABLE:=0;
    END_IF;

    (*TL23*)
    IF PL2 AND P_AL1_L_FT AND NOT PL23 THEN
      PL2:=0;
      PL23:=1;
      STABLE:=0;
    END_IF;

    (*TL2*)
    IF PL23 AND P_AL1_L_FT AND NOT PL3 THEN
      PL23:=0;
      PL3:=1;
      STABLE:=0;
    END_IF;

    (*TL3*)
    IF PL3 AND P_AL1_L_BK AND NOT PL4 AND NOT PUSH_L AND NOT P_LID THEN
      PL3:=0;
      PL4:=1;
      PUSH_L:=1;
      P_LID:=1;
      STABLE:=0;
    END_IF;

    (*TL4*)
    IF PL4 AND PLF1 AND S_AL1_L1 AND NOT PL5 THEN
      PL4:=0;
      PLF1:=0;
      PL5:=1;
      STABLE:=0;
    END_IF;

    (*TL5*)
    IF PL5 AND PLF2 AND S_AL1_L2 AND NOT PL6 AND NOT PLF1 THEN
      PL5:=0;
      PLF2:=0;
      PL6:=1;
      PLF1:=1;
      STABLE:=0;
    END_IF;

    (*TL6*)
    IF PL6 AND PLF3 AND S_AL1_L3 AND  NOT PL7 AND NOT PLF2 THEN
      PL6:=0;
      PLF3:=0;
      PL7:=1;
      PLF2:=1;
      STABLE:=0;
    END_IF;

    (*TL7*)
    IF PL7 AND PLF4 AND S_AL1_LP AND NOT PL8 THEN
      PL7:=0;
      PLF4:=0;
      PL8:=1;
      STABLE:=0;
    END_IF;

    (*TL8*)
    IF PL8 AND LP_AL1_CLAMPED AND NOT PL9 THEN
      PL8:=0;
      PL9:=1;
      STABLE:=0;
    END_IF;

    (*TL9*)
    IF PL9 AND NOT LP_AL1_CLAMPED AND NOT PLF3 AND NOT PLF4 THEN
      PL9:=0;
      PLF3:=1;
      PLF4:=1;
      STABLE:=0;
    END_IF;

  END_WHILE;

  (*============================================================*)
  (* OUTPUTS *)
  (*============================================================*)
  (*P_AL1_B*)
  IF PB2 OR PB23 THEN
    P_AL1_B:=1;
  END_IF;
  IF P_BASE OR PB1 OR PB3 THEN
    P_AL1_B:=0;
  END_IF;

  (*SB_AL1_B1*)
  IF PB5 THEN
    SB_AL1_B1:=1;
  END_IF;
  IF PBF1 THEN
    SB_AL1_B1:=0;
  END_IF;

  (*SB_AL1_B2*)
  IF PB6 THEN
    SB_AL1_B2:=1;
  END_IF;
  IF PBF2 THEN
    SB_AL1_B2:=0;
  END_IF;

  (*SB_AL1_B3*)
  IF PB7 THEN
    SB_AL1_B3:=1;
  END_IF;
  IF PBF3 THEN
    SB_AL1_B3:=0;
  END_IF;

  (*LP_AL1_CLAMP*)
  IF PB8 OR PB9 THEN
    LP_AL1_CLAMP:=1;
  END_IF;
  IF PBF4 THEN
    LP_AL1_CLAMP:=0;
  END_IF;

  (*P_AL1_L*)
  IF PL2 OR PL23 THEN
    P_AL1_L:=1;
  END_IF;
  IF P_LID OR PL1 OR PL3 THEN
    P_AL1_L:=0;
  END_IF;

  (*SB_AL1_L1*)
  IF PL5 THEN
    SB_AL1_L1:=1;
  END_IF;
  IF PLF1 THEN
    SB_AL1_L1:=0;
  END_IF;

  (*SB_AL1_L2*)
  IF PL6 THEN
    SB_AL1_L2:=1;
  END_IF;
  IF PLF2 THEN
    SB_AL1_L2:=0;
  END_IF;

  (*SB_AL1_L3*)
  IF PL7 THEN
    SB_AL1_L3:=1;
  END_IF;
  IF PLF3 THEN
    SB_AL1_L3:=0;
  END_IF;

  (*LP_AL1_CLAMP*)
  IF PL8 OR PL9 THEN
    LP_AL1_CLAMP:=1;
  END_IF;
  IF PLF4 THEN
    LP_AL1_CLAMP:=0;
  END_IF;

END_PROGRAM

CONFIGURATION Config0

  RESOURCE Res0 ON PLC
    TASK task0(INTERVAL := T#20ms,PRIORITY := 0);
    PROGRAM instance0 WITH task0 : buffer_stage;
  END_RESOURCE
END_CONFIGURATION

(* ---- lb_claude_assisted_694d1972ded0_0029.st ---- *)
FUNCTION_BLOCK GE_0
  VAR_INPUT
    IN1 : DINT;
    IN2 : DINT;
  END_VAR
  VAR_OUTPUT
    OUT : BOOL;
  END_VAR
  VAR
    mytimer : TON;
  END_VAR

  OUT:=FALSE;
  IF IN1>=IN2 then
    OUT:=TRUE;
  END_IF;

  IF mytimer.Q = TRUE THEN
      mytimer(IN := TRUE, PT := T#9999h);
  ELSE
      mytimer(IN := TRUE, PT := t#8000ms);
  END_IF;

  IF mytimer.Q = TRUE then

      OUT:=TRUE;

  End_IF;
END_FUNCTION_BLOCK

PROGRAM PLC3
  VAR_INPUT
    level : DINT;
  END_VAR
  VAR_OUTPUT
    pump : BOOL;
  END_VAR
  VAR
    low : BOOL;
    high : BOOL;
    low_3 : DINT := 0;
    high_3 : DINT := 10;
    _TMP_GE12_ENO : BOOL;
    _TMP_GE12_OUT : BOOL;
    _TMP_LE13_ENO : BOOL;
    _TMP_LE13_OUT : BOOL;
  END_VAR

  _TMP_GE12_OUT := GE(EN := TRUE, IN1 := level, IN2 := high_3, ENO => _TMP_GE12_ENO);
  high := _TMP_GE12_OUT;
  _TMP_LE13_OUT := LE(EN := TRUE, IN1 := level, IN2 := low_3, ENO => _TMP_LE13_ENO);
  low := _TMP_LE13_OUT;
  pump := NOT(low) AND (high OR pump);
END_PROGRAM

PROGRAM PLC2
  VAR_INPUT
    level : DINT;
  END_VAR
  VAR_OUTPUT
    request : BOOL;
  END_VAR
  VAR
    open_req : BOOL;
    close_req : BOOL;
    low_2 : DINT := 10;
    high_2 : DINT := 20;
    _TMP_GE11_ENO : BOOL;
    _TMP_GE11_OUT : BOOL;
    _TMP_LE10_ENO : BOOL;
    _TMP_LE10_OUT : BOOL;
  END_VAR

  _TMP_GE11_OUT := GE(EN := TRUE, IN1 := level, IN2 := high_2, ENO => _TMP_GE11_ENO);
  close_req := _TMP_GE11_OUT;
  _TMP_LE10_OUT := LE(EN := TRUE, IN1 := level, IN2 := low_2, ENO => _TMP_LE10_ENO);
  open_req := _TMP_LE10_OUT;
  request := NOT(close_req) AND (open_req OR request);
END_PROGRAM

PROGRAM PLC1
  VAR_INPUT
    level : DINT;
    request : DINT;
  END_VAR
  VAR_OUTPUT
    pumps : BOOL;
    valve : BOOL;
  END_VAR
  VAR
    low : BOOL;
    high : BOOL;
    open_req : BOOL;
    close_req : BOOL;
    low_1 : DINT := 40;
    high_1 : DINT := 80;
    GE_00 : GE_0;
    _TMP_LE3_ENO : BOOL;
    _TMP_LE3_OUT : BOOL;
    _TMP_EQ31_ENO : BOOL;
    _TMP_EQ31_OUT : BOOL;
    _TMP_EQ24_ENO : BOOL;
    _TMP_EQ24_OUT : BOOL;
  END_VAR

  _TMP_LE3_OUT := LE(EN := TRUE, IN1 := level, IN2 := low_1, ENO => _TMP_LE3_ENO);
  low := _TMP_LE3_OUT;
  GE_00(EN := TRUE, IN1 := level, IN2 := high_1);
  high := GE_00.OUT;
  pumps := NOT(high) AND (low OR pumps);
  valve := NOT(close_req) AND (valve OR open_req AND NOT(low));
  _TMP_EQ31_OUT := EQ(EN := TRUE, IN1 := request, IN2 := 1, ENO => _TMP_EQ31_ENO);
  open_req := _TMP_EQ31_OUT;
  _TMP_EQ24_OUT := EQ(EN := TRUE, IN1 := request, IN2 := 0, ENO => _TMP_EQ24_ENO);
  close_req := _TMP_EQ24_OUT;
END_PROGRAM

CONFIGURATION Config0

  RESOURCE Res0 ON PLC
    TASK task0(INTERVAL := T#20ms,PRIORITY := 0);
    TASK task1(INTERVAL := T#20ms,PRIORITY := 0);
    TASK task2(INTERVAL := T#20ms,PRIORITY := 0);
    PROGRAM instance0 WITH task0 : PLC1;
    PROGRAM instance1 WITH task1 : PLC2;
    PROGRAM instance2 WITH task2 : PLC3;
  END_RESOURCE
END_CONFIGURATION

(* ---- lb_claude_assisted_6a5538546aea_0005.st ---- *)
FUNCTION_BLOCK rand_generator
  VAR_INPUT
    IN : BOOL;
  END_VAR
  VAR
    M : BOOL;
    INIT : BOOL;
  END_VAR
  VAR_OUTPUT
    RANDOM : INT := 0;
    BOTTKO : INT := 0;
    BOTTOK : INT := 0;
  END_VAR

  IF INIT = 0 THEN
    {srand(time(NULL))}
    INIT := 1;
  END_IF;

  IF M = 0 AND IN = 1 THEN
    {int r = rand() % 10;
    SetFbVar(RANDOM,r)}
    IF RANDOM = 0 THEN
      {int bKo = 0;
      bKo = GetFbVar(BOTTKO);
      bKo++;
      SetFbVar(BOTTKO,bKo)}
    ELSE
      {int bOk = 0;
      bOk = GetFbVar(BOTTOK);
      bOk++;
      SetFbVar(BOTTOK,bOk)}
    END_IF;
  END_IF;
  M := IN;
END_FUNCTION_BLOCK

PROGRAM BeerFactory
  VAR
    InputSegnale AT %QX0.0 : BOOL;
    SensorePosBott AT %QX0.1 : BOOL;
    MotoreCarrello AT %QX0.2 : BOOL;
    MotoreDistribuzione AT %QX0.3 : BOOL;
    SensoreLimite AT %QX0.4 : BOOL;
    NumeroMaxBott AT %IW0 : INT := 32767;
    NumeroBott AT %QW0 : INT := 0;
    NumeroRand AT %QW1 : INT := 0;
    NumBottKo AT %QW2 : INT := 0;
    NumBottOk AT %QW3 : INT := 0;
    Count AT %IX0.0 : BOOL;
  END_VAR
  VAR
    EsCarrello : TP;
    EsDistribu : TP;
    RestartCarrello : TP;
    ContatoreBott : CTU;
    rand_generator0 : rand_generator;
    R_TRIG1 : R_TRIG;
  END_VAR

  EsCarrello(IN := NOT(SensorePosBott) AND InputSegnale, PT := T#5s);
  MotoreCarrello := EsCarrello.Q;
  SensorePosBott := NOT(MotoreCarrello) AND InputSegnale;
  MotoreDistribuzione := NOT(MotoreCarrello) AND InputSegnale;
  EsDistribu(IN := NOT(MotoreCarrello) AND InputSegnale, PT := T#5s);
  SensoreLimite := EsDistribu.Q;
  IF NOT(MotoreCarrello) AND NOT(SensoreLimite) AND InputSegnale THEN
      RestartCarrello(IN := NOT(MotoreCarrello) AND NOT(SensoreLimite) AND InputSegnale, PT := T#9999h);
  ELSE
      RestartCarrello(IN := NOT(MotoreCarrello) AND NOT(SensoreLimite) AND InputSegnale, PT := T#1s);
  END_IF;
  SensorePosBott := RestartCarrello.Q;
  R_TRIG1(CLK := RestartCarrello.Q);
  ContatoreBott(CU := R_TRIG1.Q, PV := NumeroMaxBott);
  Count := ContatoreBott.Q;
  NumeroBott := ContatoreBott.CV;
  rand_generator0(IN := RestartCarrello.Q);
  NumeroRand := rand_generator0.RANDOM;
  NumBottKo := rand_generator0.BOTTKO;
  NumBottOk := rand_generator0.BOTTOK;
END_PROGRAM

CONFIGURATION Config0

  RESOURCE Res0 ON PLC
    TASK task0(INTERVAL := T#20ms,PRIORITY := 0);
    PROGRAM instance0 WITH task0 : BeerFactory;
  END_RESOURCE
END_CONFIGURATION

(* ---- lb_claude_assisted_6c2e20ba6a85_0038.st ---- *)
FUNCTION_BLOCK rand_generator
  VAR_INPUT
    IN : BOOL;
  END_VAR
  VAR
    M : BOOL;
    INIT : BOOL;
  END_VAR
  VAR_OUTPUT
    RANDOM : INT := 0;
    BOTTKO : INT := 0;
    BOTTOK : INT := 0;
  END_VAR

  IF INIT = 0 THEN
    {srand(time_t(NULL))}
    INIT := 1;
  END_IF;

  IF M = 0 AND IN = 1 THEN
    {int r = rand() % 10;
    SetFbVar(RANDOM,r)}
    IF RANDOM = 0 THEN
      {int bKo = 0;
      bKo = GetFbVar(BOTTKO);
      bKo++;
      SetFbVar(BOTTKO,bKo)}
    ELSE
      {int bOk = 0;
      bOk = GetFbVar(BOTTOK);
      bOk++;
      SetFbVar(BOTTOK,bOk)}
    END_IF;
  END_IF;
  M := IN;
END_FUNCTION_BLOCK

PROGRAM BeerFactory
  VAR
    InputSegnale AT %QX0.0 : BOOL;
    SensorePosBott AT %QX0.1 : BOOL;
    MotoreCarrello AT %QX0.2 : BOOL;
    MotoreDistribuzione AT %QX0.3 : BOOL;
    SensoreLimite AT %QX0.4 : BOOL;
    NumeroMaxBott AT %IW0 : INT := 32767;
    NumeroBott AT %QW0 : INT := 0;
    NumeroRand AT %QW1 : INT := 0;
    NumBottKo AT %QW2 : INT := 0;
    NumBottOk AT %QW3 : INT := 0;
    Count AT %IX0.0 : BOOL;
  END_VAR
  VAR
    EsCarrello : TP;
    EsDistribu : TP;
    RestartCarrello : TP;
    ContatoreBott : CTU;
    rand_generator0 : rand_generator;
    R_TRIG1 : R_TRIG;
  END_VAR

  EsCarrello(IN := NOT(SensorePosBott) AND InputSegnale, PT := T#5s);
  MotoreCarrello := EsCarrello.Q;
  SensorePosBott := NOT(MotoreCarrello) AND InputSegnale;
  MotoreDistribuzione := NOT(MotoreCarrello) AND InputSegnale;
  IF NOT(MotoreCarrello) AND NOT(SensoreLimite) AND InputSegnale THEN
      EsDistribu(IN := NOT(MotoreCarrello) AND InputSegnale, PT := T#9999h);
  ELSE
      EsDistribu(IN := NOT(MotoreCarrello) AND InputSegnale, PT := T#5s);
  END_IF;
  SensoreLimite := EsDistribu.Q;
  RestartCarrello(IN := NOT(MotoreCarrello) AND NOT(SensoreLimite) AND InputSegnale, PT := T#1s);
  SensorePosBott := RestartCarrello.Q;
  R_TRIG1(CLK := RestartCarrello.Q);
  ContatoreBott(CU := R_TRIG1.Q, PV := NumeroMaxBott);
  Count := ContatoreBott.Q;
  NumeroBott := ContatoreBott.CV;
  rand_generator0(IN := RestartCarrello.Q);
  NumeroRand := rand_generator0.RANDOM;
  NumBottKo := rand_generator0.BOTTKO;
  NumBottOk := rand_generator0.BOTTOK;
END_PROGRAM

CONFIGURATION Config0

  RESOURCE Res0 ON PLC
    TASK task0(INTERVAL := T#20ms,PRIORITY := 0);
    PROGRAM instance0 WITH task0 : BeerFactory;
  END_RESOURCE
END_CONFIGURATION

(* ---- lb_claude_assisted_6c400fd06623_0016.st ---- *)
(*
This code implements a randomly grown symbolic expression:

(((xor(xor((xor(xor(xor(xor(IN19, (!(IN48 | IN21)) & (!(xor(xor(IN30, IN18), IN5)))), IN21), ((xor(xor(IN23 | IN7, IN44 | IN43), IN28 & IN45)) & ((!(IN4)) | (IN37 | IN4))) | (xor(xor((IN10 | IN19) | (IN27 & IN18), IN45), !(IN41)))), IN21)) & ((((IN36 | false) | ((!(IN22)) | (xor(xor(IN17, IN20), IN45)))) | (((xor(xor(IN40, IN49), IN35)) & (!(IN19))) & (xor(xor(xor(xor(IN32, IN22), IN46), !(IN2)), xor(xor(IN46, IN23), IN28))))) | ((((IN7 & IN47) & (IN5 & IN32)) & ((IN29 | IN13) | (true & IN42))) & ((true & (IN8 & IN29)) & (xor(xor(!(IN46), !(IN24)), xor(xor(IN6, IN16), IN4)))))), (((!(!(IN20 | IN46))) | (!(xor(xor(!(IN16), xor(xor(IN12, IN9), IN4)), IN31 | IN40)))) & IN49) & (xor(xor(IN41, (xor(xor((xor(xor(true, IN18), false)) & (xor(xor(IN10, IN15), IN4)), (!(IN14)) & IN12), (IN43 | IN32) & IN32)) & (IN31 | ((xor(xor(IN22, true), IN17)) | (xor(xor(IN49, IN20), false))))), xor(xor(!(IN45), IN46), IN2 | (xor(xor(IN11, IN2 & IN18), IN43 | IN11)))))), IN11)) | IN13) | (xor(xor(xor(xor((!((!((IN29 | IN7) & (IN48 | IN42))) | IN20)) | (!(IN21)), (xor(xor(xor(xor(xor(xor((xor(xor(IN1, IN10), IN29)) | (IN2 & IN25), xor(xor(xor(xor(IN34, IN6), IN25), IN41 & IN10), IN36 & IN25)), (IN6 & IN20) | (IN47 | IN26)), IN7), !((IN43 & IN25) | (xor(xor(IN44, IN44), IN30)))), IN15 | (IN8 & (xor(xor(xor(xor(IN3, IN16), IN33), IN3 & IN40), !(IN40))))), IN31 & IN19)) & (IN27 & (!(IN47 & (xor(xor(IN5, IN38 & IN40), IN30)))))), xor(xor(((!(!(IN24))) & (xor(xor(IN30, IN2), xor(xor(xor(xor(IN38, true), IN8), IN33 & IN9), xor(xor(IN49, IN40), IN43))))) & (((true & (xor(xor(IN49, IN36), IN7))) | ((!(IN21)) | (IN4 & IN40))) & IN47), ((((IN13 | IN3) & IN30) & (xor(xor(IN3 & IN14, !(IN41)), !(IN22)))) & ((!(IN33 | IN21)) | (!(IN18 & IN42)))) | (xor(xor((xor(xor(!(IN37), IN49 | IN14), IN42)) & (!(IN1 & IN30)), ((!(IN18)) & (xor(xor(IN28, IN28), IN42))) & (IN40 | IN32)), !(IN34 & (xor(xor(IN45, IN21), IN18)))))), xor(xor(!(!(xor(xor(IN48 | IN1, !(IN12)), !(IN27)))), ((xor(xor(IN43 | IN15, IN9 | IN20), xor(xor(IN4, IN4), IN11))) & IN35) & (IN21 | (!(IN13 & IN21)))), ((xor(xor(xor(xor(IN29, IN17), IN6), IN23 | IN2), IN46 | IN28)) & (!(IN42))) | IN9))), xor(xor(IN21, !(!(!(!((xor(xor(IN47, IN29), IN31)) & (IN3 & IN43)))))), (!((xor(xor(!(IN27 | IN39), xor(xor(xor(xor(IN1, IN14), IN16), false | IN8), IN47 | IN1)), xor(xor(IN36 & IN31, !(IN39)), IN44 | IN33))) & ((IN8 | (IN5 | IN34)) & (!(xor(xor(IN12, IN31), IN12)))))) | ((((!(xor(xor(IN45, IN8), IN46))) & IN45) & IN8) | (!(!((IN28 & IN42) & (IN50 | IN35))))))), xor(xor(IN29, !((IN34 | (IN1 | (IN12 & (IN6 | IN15)))) & ((!(!(IN32 & IN18))) & (!(!(IN6 & IN28)))))), ((!(!(IN25))) | (xor(xor(xor(xor(!(IN3 & IN34), xor(xor(IN16 & IN26, !(IN26)), IN17)), (IN33 & IN37) & (!(IN32))), ((IN38 | IN8) & (!(IN19))) | (xor(xor(!(IN29), IN4 | IN21), IN39 & IN36))), (xor(xor(IN41 | IN43, xor(xor(IN32, IN10), IN28)), IN18 & IN1)) | (IN25 & IN34)))) & IN8)))) | IN13

*)

FUNCTION_BLOCK F_CollectInput
  VAR_IN_OUT
      Data : ARRAY[1..50] OF BOOL;
  END_VAR
  VAR_INPUT
      TICK  : BOOL := 0;
      IN1   : BOOL := 0;
      IN2   : BOOL := 0;
      IN3   : BOOL := 0;
      IN4   : BOOL := 0;
      IN5   : BOOL := 0;
      RESET : BOOL := FALSE;
  END_VAR
  VAR_OUTPUT
      Finished : BOOL;
  END_VAR
  VAR
      j    : USINT := 1;
      tock : BOOL  := 0;
  END_VAR
  IF NOT RESET AND tock = NOT TICK THEN
      Data[j]   := IN1;
      Data[j+1] := IN2;
      Data[j+2] := IN3;
      Data[j+3] := IN4;
      Data[j+4] := IN5;
      j := j + 5;
      tock := TICK;
  ELSE
      j := 1;
      tock := 0;
  END_IF;
  Finished := (j > 50);
END_FUNCTION_BLOCK

PROGRAM Boiler
  VAR
    Data  : ARRAY[1..50] OF BOOL;
    Ready : BOOL;
    CollectInput : F_CollectInput;
  END_VAR
  VAR
    TICK     AT %IX1.0 : BOOL;
    IN1      AT %IX0.3 : BOOL;
    IN2      AT %IX0.4 : BOOL;
    IN3      AT %IX0.5 : BOOL;
    IN4      AT %IX0.6 : BOOL;
    IN5      AT %IX0.7 : BOOL;
    OutReady AT %QX0.0 : BOOL := FALSE;
    FeedNext AT %QX0.1 : BOOL := FALSE;
    Out      AT %QX0.2 : BOOL;
  END_VAR
  CollectInput(TICK:=TICK, IN1:=IN1, IN2:=IN2, IN3:=IN3, IN4:=IN4, IN5:=IN5);
  Ready := CollectInput.Finished;
  FeedNext := 1;
  IF Ready THEN
    Out := ((((((((((Data[19] XOR ((NOT (Data[48] OR Data[21])) AND (NOT ((Data[30] XOR Data[18]) XOR Data[5])))) XOR Data[21]) XOR (((((Data[23] OR Data[7]) XOR (Data[44] OR Data[43])) XOR (Data[28] AND Data[45])) AND ((NOT Data[4]) OR (Data[37] OR Data[4]))) OR ((((Data[10] OR Data[19]) OR (Data[27] AND Data[18])) XOR Data[45]) XOR (NOT Data[41])))) XOR Data[21]) AND ((((Data[36] OR FALSE) OR ((NOT Data[22]) OR ((Data[17] XOR Data[20]) XOR Data[45]))) OR ((((Data[40] XOR Data[49]) XOR Data[35]) AND (NOT Data[19])) AND ((((Data[32] XOR Data[22]) XOR Data[46]) XOR (NOT Data[2])) XOR ((Data[46] XOR Data[23]) XOR Data[28])))) OR ((((Data[7] AND Data[47]) AND (Data[5] AND Data[32])) AND ((Data[29] OR Data[13]) OR (TRUE AND Data[42]))) AND ((TRUE AND (Data[8] AND Data[29])) AND (((NOT Data[46]) XOR (NOT Data[24])) XOR ((Data[6] XOR Data[16]) XOR Data[4])))))) XOR ((((NOT (NOT (Data[20] OR Data[46]))) OR (NOT (((NOT Data[16]) XOR ((Data[12] XOR Data[9]) XOR Data[4])) XOR (Data[31] OR Data[40])))) AND Data[49]) AND ((Data[41] XOR ((((((TRUE XOR Data[18]) XOR FALSE) AND ((Data[10] XOR Data[15]) XOR Data[4])) XOR ((NOT Data[14]) AND Data[12])) XOR ((Data[43] OR Data[32]) AND Data[32])) AND (Data[31] OR (((Data[22] XOR TRUE) XOR Data[17]) OR ((Data[49] XOR Data[20]) XOR FALSE))))) XOR (((NOT Data[45]) XOR Data[46]) XOR (Data[2] OR ((Data[11] XOR (Data[2] AND Data[18])) XOR (Data[43] OR Data[11]))))))) XOR Data[11]) OR Data[13]) OR ((((((NOT ((NOT ((Data[29] OR Data[7]) AND (Data[48] OR Data[42]))) OR Data[20])) OR (NOT Data[21])) XOR ((((((((((Data[1] XOR Data[10]) XOR Data[29]) OR (Data[2] AND Data[25])) XOR ((((Data[34] XOR Data[6]) XOR Data[25]) XOR (Data[41] AND Data[10])) XOR (Data[36] AND Data[25]))) XOR ((Data[6] AND Data[20]) OR (Data[47] OR Data[26]))) XOR Data[7]) XOR (NOT ((Data[43] AND Data[25]) OR ((Data[44] XOR Data[44]) XOR Data[30])))) XOR (Data[15] OR (Data[8] AND ((((Data[3] XOR Data[16]) XOR Data[33]) XOR (Data[3] AND Data[40])) XOR (NOT Data[40]))))) XOR (Data[31] AND Data[19])) AND (Data[27] AND (NOT (Data[47] AND ((Data[5] XOR (Data[38] AND Data[40])) XOR Data[30])))))) XOR (((((NOT (NOT Data[24])) AND ((Data[30] XOR Data[2]) XOR ((((Data[38] XOR TRUE) XOR Data[8]) XOR (Data[33] AND Data[9])) XOR ((Data[49] XOR Data[40]) XOR Data[43])))) AND (((TRUE AND ((Data[49] XOR Data[36]) XOR Data[7])) OR ((NOT Data[21]) OR (Data[4] AND Data[40]))) AND Data[47])) XOR (((((Data[13] OR Data[3]) AND Data[30]) AND (((Data[3] AND Data[14]) XOR (NOT Data[41])) XOR (NOT Data[22]))) AND ((NOT (Data[33] OR Data[21])) OR (NOT (Data[18] AND Data[42])))) OR ((((((NOT Data[37]) XOR (Data[49] OR Data[14])) XOR Data[42]) AND (NOT (Data[1] AND Data[30]))) XOR (((NOT Data[18]) AND ((Data[28] XOR Data[28]) XOR Data[42])) AND (Data[40] OR Data[32]))) XOR (NOT (Data[34] AND ((Data[45] XOR Data[21]) XOR Data[18])))))) XOR (((NOT (NOT (((Data[48] OR Data[1]) XOR (NOT Data[12])) XOR (NOT Data[27])))) XOR (((((Data[43] OR Data[15]) XOR (Data[9] OR Data[20])) XOR ((Data[4] XOR Data[4]) XOR Data[11])) AND Data[35]) AND (Data[21] OR (NOT (Data[13] AND Data[21]))))) XOR ((((((Data[29] XOR Data[17]) XOR Data[6]) XOR (Data[23] OR Data[2])) XOR (Data[46] OR Data[28])) AND (NOT Data[42])) OR Data[9])))) XOR ((Data[21] XOR (NOT (NOT (NOT (NOT (((Data[47] XOR Data[29]) XOR Data[31]) AND (Data[3] AND Data[43]))))))) XOR ((NOT ((((NOT (Data[27] OR Data[39])) XOR ((((Data[1] XOR Data[14]) XOR Data[16]) XOR (FALSE OR Data[8])) XOR (Data[47] OR Data[1]))) XOR (((Data[36] AND Data[31]) XOR (NOT Data[39])) XOR (Data[44] OR Data[33]))) AND ((Data[8] OR (Data[5] OR Data[34])) AND (NOT ((Data[12] XOR Data[31]) XOR Data[12]))))) OR ((((NOT ((Data[45] XOR Data[8]) XOR Data[46])) AND Data[45]) AND Data[8]) OR (NOT (NOT ((Data[28] AND Data[42]) AND (Data[50] OR Data[35])))))))) XOR ((Data[29] XOR (NOT ((Data[34] OR (Data[1] OR (Data[12] AND (Data[6] OR Data[15])))) AND ((NOT (NOT (Data[32] AND Data[18]))) AND (NOT (NOT (Data[6] AND Data[28]))))))) XOR (((NOT (NOT Data[25])) OR (((((NOT (Data[3] AND Data[34])) XOR (((Data[16] AND Data[26]) XOR (NOT Data[26])) XOR Data[17])) XOR ((Data[33] AND Data[37]) AND (NOT Data[32]))) XOR (((Data[38] OR Data[8]) AND (NOT Data[19])) OR (((NOT Data[29]) XOR (Data[4] OR Data[21])) XOR (Data[39] AND Data[36])))) XOR ((((Data[41] OR Data[43]) XOR ((Data[32] XOR Data[10]) XOR Data[28])) XOR (Data[18] AND Data[1])) OR (Data[25] AND Data[34])))) AND Data[8])))) OR Data[13]);
    IF Ready THEN
        OutReady := 0;
    ELSE
        OutReady := 1;
    END_IF;
    CollectInput(RESET:=TRUE);
  END_IF;
END_PROGRAM

CONFIGURATION Config0
  RESOURCE Res0 ON PLC
    TASK task0(INTERVAL := T#20ms,PRIORITY := 0);
    PROGRAM instance0 WITH task0 : Boiler;
  END_RESOURCE
END_CONFIGURATION

(* ---- lb_claude_assisted_6ec6facc7008_0015.st ---- *)
FUNCTION UDINT_TO_TIME2:TIME
	VAR_INPUT
		IN :	UDINT;
	END_VAR
	UDINT_TO_TIME2 := DINT_TO_TIME(UDINT_TO_DINT(IN));
END_FUNCTION

FUNCTION_BLOCK T_PLC_MS_block
	VAR_OUTPUT
		T_PLC_MS :	UDINT;
	END_VAR

	VAR_EXTERNAL
		PLC_TICKS_PER_SEC :	INT;
		PLC_SYS_TICK_CNT :	DINT;
	END_VAR

	VAR
		debug :	BOOL;(*Debug-Mode ON / OFF*)
		N :	INT;(*Debug-Faktor*)
		Offset :	UDINT;(*Debug-Offset*)
		temp :	DWORD := DWORD#1;(*Debug-Offset*)
		mode :	BOOL;(*modus*)
		faktor :	UDINT;(*Systemtakt-Faktor*)
		init :	BOOL;
		v_plc_ticks_per_sec :	UDINT;
		base :	UDINT := UDINT#1000;
	END_VAR

	IF init = FALSE THEN
		v_plc_ticks_per_sec := INT_TO_UDINT(PLC_TICKS_PER_SEC);
		IF v_plc_ticks_per_sec = UDINT#1024 THEN
			faktor := UDINT#1;
			mode := FALSE;
		ELSIF v_plc_ticks_per_sec > UDINT#0 THEN
			IF v_plc_ticks_per_sec <= base THEN
				faktor := base / v_plc_ticks_per_sec;
				mode := FALSE;
			ELSE
				faktor := v_plc_ticks_per_sec / base;
				mode := TRUE;
			END_IF;
		ELSE
			faktor := UDINT#1;
		END_IF;
		init := TRUE;
	END_IF;

	IF mode THEN
		T_PLC_MS := DINT_TO_UDINT(PLC_SYS_TICK_CNT) / faktor;
	ELSE
		T_PLC_MS := DINT_TO_UDINT(PLC_SYS_TICK_CNT) * faktor;
	END_IF;

	IF debug THEN
		T_PLC_MS := (DWORD_TO_UDINT(SHL(UDINT_TO_DWORD(T_PLC_MS),N) OR SHL(temp,N)) - UDINT#1) + Offset;
	END_IF;

END_FUNCTION_BLOCK

TYPE
	oscat_ARRAY_X               : ARRAY [0..1]    OF REAL;
	oscat_XY                    : ARRAY [1..20]   OF oscat_ARRAY_X := [0,0,0,0,0,0,0,0,0,0,0,0,0,0,0,0,0,0,0,0];
END_TYPE

FUNCTION_BLOCK LINEAR_INT_Block

	VAR_INPUT
		X :	REAL;
		XY :	oscat_XY;
		PTS :	INT;
	END_VAR

	VAR_OUTPUT
		LINEAR_INT :	REAL;
	END_VAR

	VAR
		i :	INT;
		i2 :	INT;
	END_VAR

	pts := MIN(pts,20);

	i := 2;

	WHILE (i < pts) AND (XY[i][0] < X) DO
		i := i + 1;
	END_WHILE;

	i2 := i-1;

	LINEAR_INT := ((XY[i][1] - XY[i2][1]) * X - XY[i][1] * XY[i2][0] + XY[i2][1] * XY[i][0]) / (XY[i][0] - XY[i2][0]);

END_FUNCTION_BLOCK

FUNCTION_BLOCK WATER_ENTHALPY_Block

    VAR_INPUT
        T :	REAL;
    END_VAR

    VAR_OUTPUT
        RESULT :	REAL;
    END_VAR

    VAR
        Pts :	INT;
        data :	oscat_XY;
        FB_LINEAR_INT :	LINEAR_INT_Block;
    END_VAR

    IF Pts = 0 THEN
        Pts := 11;
        data[01][0] := REAL#0.0;
        data[01][1] := REAL#0.06;
        data[02][0] := REAL#10.0;
        data[02][1] := REAL#42.1;
        data[03][0] := REAL#20.0;
        data[03][1] := REAL#83.9;
        data[04][0] := REAL#30.0;
        data[04][1] := REAL#125.8;
        data[05][0] := REAL#40.0;
        data[05][1] := REAL#167.58;
        data[06][0] := REAL#50.0;
        data[06][1] := REAL#209.4;
        data[07][0] := REAL#60.0;
        data[07][1] := REAL#251.2;
        data[08][0] := REAL#70.0;
        data[08][1] := REAL#293.1;
        data[09][0] := REAL#80.0;
        data[09][1] := REAL#335.0;
        data[10][0] := REAL#90.0;
        data[10][1] := REAL#377.0;
        data[11][0] := REAL#100.0;
        data[11][1] := REAL#419.1;
    END_IF;

    FB_LINEAR_INT(X:=T,XY:=Data,Pts:=Pts);
    Result :=FB_LINEAR_INT.LINEAR_INT;

END_FUNCTION_BLOCK

FUNCTION_BLOCK R2_SET_Block

	VAR_INPUT
		X :	REAL;
	END_VAR

	VAR_OUTPUT
		R2_SET :	REAL2;
	END_VAR

	R2_SET.RX := X;
	R2_SET.R1 := 0.0;

END_FUNCTION_BLOCK

FUNCTION_BLOCK R2_ADD_Block

	VAR_INPUT
		X :	REAL2;
		Y :	REAL;
	END_VAR

	VAR_OUTPUT
		R2_ADD :	REAL2;
	END_VAR

	VAR
		temp :	REAL;
	END_VAR

	temp := X.RX;
	R2_ADD.RX := Y + X.R1 + X.RX;
	R2_ADD.R1 := temp - R2_ADD.RX + Y + X.R1;

END_FUNCTION_BLOCK

TYPE REAL2:

	STRUCT
		R1 : REAL;
		RX : REAL;
	END_STRUCT;

END_TYPE

FUNCTION_BLOCK INTEGRATE

	VAR_INPUT
		E :	BOOL := TRUE;
		X :	REAL;
		K :	REAL := 1.0;
	END_VAR

	VAR_IN_OUT
		Y :	REAL;
	END_VAR

	VAR
		X_last :	REAL;
		init :	BOOL;
		T_PLC_MS :	T_PLC_MS_block;
		last :	UDINT;
		tx :	UDINT;
	END_VAR

	T_PLC_MS();
	tx:= T_PLC_MS.T_PLC_MS;

	IF NOT init THEN
		init := TRUE;
		X_last := X;
	ELSIF E THEN
		Y := (X + X_LAST) * 0.5E-3 * UDINT_TO_REAL(tx-last) * K + Y;
		X_last := X;
	END_IF;
	last := tx;

END_FUNCTION_BLOCK

FUNCTION_BLOCK FT_INT2_Block

	VAR_INPUT
		IN :	REAL;
		K :	REAL := 1.0;
		RUN :	BOOL := TRUE;
		RST :	BOOL;
		OUT_MIN :	REAL := REAL#-1.0E-37;
		OUT_MAX :	REAL := REAL#1.0E37;
	END_VAR

	VAR_OUTPUT
		OUT :	REAL;
		LIM :	BOOL;
	END_VAR

	VAR
		integ :	INTEGRATE;
		ix :	REAL;
		val :	REAL2;
		R2_ADD :	R2_ADD_Block;
		R2_SET :	R2_SET_Block;
	END_VAR

	IF RST THEN
		R2_SET(X:=0.0);
		val:=R2_SET.R2_SET;
		out := 0.0;
	ELSE
		integ(X := IN, E := RUN, K := K, Y := ix);
		ix := integ.Y;
		R2_ADD(X:=val,Y:=ix);
		val:=R2_ADD.R2_ADD;
		ix := 0.0;
		OUT := val.RX;
	END_IF;

	(* check output for limits *)
	IF out > OUT_MIN AND out < OUT_MAX THEN
		LIM := FALSE;
	ELSE
		OUT := LIMIT(OUT_MIN, OUT, OUT_MAX);
		R2_SET(X:=OUT);
		val:=R2_SET.R2_SET;
		LIM := TRUE;
	END_IF;

END_FUNCTION_BLOCK

FUNCTION WATER_DENSITY:REAL

    VAR_INPUT
        T :	REAL;
        SAT :	BOOL;
    END_VAR

    VAR
        T2 :	REAL;
        T4 :	REAL;
    END_VAR

    T2 := T * T;
    T4 := T2 * T2;
    WATER_DENSITY := (999.83952 + 16.952577*T + -7.9905127E-3*T2 + -4.6241757E-5*T2*T + 1.0584601E-7*T4 + -2.8103006E-10*T4*T) / (1.0 + 0.0168872*T);
    IF sat THEN WATER_DENSITY := WATER_DENSITY - 0.004612 + 0.000106 * T; END_IF;

END_FUNCTION

FUNCTION TIME_TO_UDINT2:UDINT
	VAR_INPUT
		X :	TIME;
	END_VAR

	TIME_TO_UDINT2 := DINT_TO_UDINT(TIME_TO_DINT(X));
END_FUNCTION

FUNCTION_BLOCK HEAT_METER_Block

	VAR_INPUT
		TF :	REAL;
		TR :	REAL;
		LPH :	REAL;
		E :	BOOL;
		RST :	BOOL;
		CP :	REAL;
		DENSITY :	REAL;
		CONTENT :	REAL;
		PULSE_MODE :	BOOL;
		RETURN_METER :	BOOL;
		AVG_TIME :	TIME := T#5s;
	END_VAR

	VAR_OUTPUT
		C :	REAL;
	END_VAR

	VAR_IN_OUT
		Y :	REAL;
	END_VAR

	VAR
		tx :	UDINT;
		last :	UDINT;
		int1 :	FT_INT2_Block;
		edge :	BOOL;
		x :	REAL;
		init :	BOOL;
		Y_last :	REAL;
		T_PLC_MS :	T_PLC_MS_Block;
		WATER_ENTHALPY :	WATER_ENTHALPY_Block;
		wa_TF :	REAL;
		wa_TR :	REAL;
	END_VAR

	IF rst THEN
		int1(rst := TRUE);
		int1.rst := FALSE;
		C := 0.0;
		Y := 0.0;
	ELSIF e THEN
		water_enthalpy(T:=TF);
		wa_TF:=water_enthalpy.Result;

		water_enthalpy(T:=TR);
		wa_TR:=water_enthalpy.Result;

		X := (WATER_DENSITY(SEL(return_meter, TF, TR), FALSE) * (wa_TF - wa_TR) * (1.0 - content) + CP * Density * content * (TF-TR));
	END_IF;

	int1(run := NOT pulse_mode AND e, in := X * LPH * 2.77777777777E-4);
	IF pulse_mode THEN
		IF NOT edge AND E THEN Y := Y + X * LPH; END_IF;
	ELSE
		Y := int1.Out;
	END_IF;

	edge := e;

	T_PLC_MS();
	tx:= T_PLC_MS.T_PLC_MS;

	IF NOT init THEN
		init := TRUE;
		last := tx;
	END_IF;

	IF (tx - last >= TIME_TO_UDINT2(AVG_TIME)) AND (avg_time > T#0s) THEN
		last := tx;
		IF tx - last >= TIME_TO_UDINT2(AVG_TIME) AND avg_time > T#0s THEN
		    C := 0.0;
		ELSE
		    C := (Y - Y_last) * 3.6E12 / TIME_TO_REAL(AVG_TIME);
		END_IF;
		Y_last := Y;
	END_IF;

END_FUNCTION_BLOCK

PROGRAM program0
	VAR
	    TF :	REAL;
		TR :	REAL;
		LPH :	REAL;
		E :	BOOL;
		RST :	BOOL;
		CP :	REAL;
		DENSITY :	REAL;
		CONTENT :	REAL;
		PULSE_MODE :	BOOL;
		RETURN_METER :	BOOL;
		AVG_TIME :	TIME := T#5s;
		Y :	REAL;
		C :	REAL;

		func_block : HEAT_METER_Block;
  	END_VAR
	func_block.TF := TF;
	func_block.TR := TR;
	func_block.LPH := LPH;
	func_block.E := E;
	func_block.RST := RST;
	func_block.CP := CP;
	func_block.DENSITY := DENSITY;
	func_block.CONTENT := CONTENT;
	func_block.PULSE_MODE := PULSE_MODE;
	func_block.RETURN_METER := RETURN_METER;
	func_block.AVG_TIME := AVG_TIME;
	func_block.Y := Y;

	func_block();
	Y := func_block.Y;
	C := func_block.C;
END_PROGRAM

CONFIGURATION Config0
	VAR_GLOBAL
		PLC_TICKS_PER_SEC :	INT;
		PLC_SYS_TICK_CNT :	DINT;
	END_VAR
  	RESOURCE Res0 ON PLC
    	TASK task0(INTERVAL := T#20ms,PRIORITY := 0);
    	PROGRAM instance0 WITH task0 : program0;
  	END_RESOURCE
END_CONFIGURATION

(* ---- lb_claude_assisted_6f944b9ecc8c_0030.st ---- *)
FUNCTION UDINT_TO_TIME2:TIME

	VAR_INPUT
		IN :	UDINT;
	END_VAR

	UDINT_TO_TIME2 := DINT_TO_TIME(UDINT_TO_DINT(IN));

END_FUNCTION

FUNCTION_BLOCK T_PLC_MS_block
	VAR_OUTPUT
		T_PLC_MS :	UDINT;
	END_VAR

	VAR
		PLC_TICKS_PER_SEC :	INT;
		PLC_SYS_TICK_CNT :	DINT;
	END_VAR

	VAR
		debug :	BOOL;(*Debug-Mode ON / OFF*)
		N :	INT;(*Debug-Faktor*)
		Offset :	UDINT;(*Debug-Offset*)
		temp :	DWORD := DWORD#1;(*Debug-Offset*)
		MODE :	BOOL;(*modus*)
		faktor :	UDINT;(*Systemtakt-Faktor*)
		init :	BOOL;
		v_plc_ticks_per_sec :	UDINT;
		base :	UDINT := UDINT#1000;
	END_VAR

	IF init = FALSE THEN
		v_plc_ticks_per_sec := INT_TO_UDINT(PLC_TICKS_PER_SEC);
		IF v_plc_ticks_per_sec = UDINT#1024 THEN
			faktor := UDINT#1;
			MODE := FALSE;
		ELSIF v_plc_ticks_per_sec > UDINT#0 THEN
			IF v_plc_ticks_per_sec <= base THEN
				faktor := base / v_plc_ticks_per_sec;
				MODE := FALSE;
			ELSE
				faktor := v_plc_ticks_per_sec / base;
				MODE := TRUE;
			END_IF;
		ELSE
			faktor := UDINT#1;
		END_IF;
		init := TRUE;
	END_IF;

	IF MODE THEN
		T_PLC_MS := DINT_TO_UDINT(PLC_SYS_TICK_CNT) / faktor;
	ELSE
		T_PLC_MS := DINT_TO_UDINT(PLC_SYS_TICK_CNT) * faktor;
	END_IF;

	IF debug THEN
		T_PLC_MS := (DWORD_TO_UDINT(SHL(UDINT_TO_DWORD(T_PLC_MS),N) OR SHL(temp,N)) - UDINT#1) + Offset;
	END_IF;
END_FUNCTION_BLOCK

FUNCTION TIME_TO_UDINT2:UDINT
	VAR_INPUT
		X :	TIME;
	END_VAR

	TIME_TO_UDINT2 := DINT_TO_UDINT(TIME_TO_DINT(X));
END_FUNCTION

FUNCTION_BLOCK ACTUATOR_COIL_Block

	VAR_INPUT
		IN :	BOOL;
		SELF_ACT_CYCLE :	TIME := T#10d;
		SELF_ACT_TIME :	TIME := T#1s;
	END_VAR

	VAR_OUTPUT
		OUT :	BOOL;
		STATUS :	BYTE;
	END_VAR

	VAR
		last :	UDINT;
		init :	BOOL;
		TX :	UDINT;
		now :	UDINT;
		T_PLC_MS :	T_PLC_MS_block;
	END_VAR

	T_PLC_MS();
	now := T_PLC_MS.T_PLC_MS;

	IF NOT init THEN
		last := now;
		init := TRUE;
	ELSIF IN THEN
		OUT := TRUE;
		STATUS := BYTE#101;
		LAST := now;
	ELSE
		OUT := FALSE;
		STATUS := BYTE#100;
		TX := now - last;
		IF (self_act_cycle > T#0s) AND (TX >= TIME_TO_UDINT2(self_act_cycle)) THEN
			OUT := TRUE;
			IF (self_act_cycle > T#0s) AND (TX >= TIME_TO_UDINT2(self_act_cycle)) THEN
			    STATUS := BYTE#101;
			ELSE
			    STATUS := BYTE#102;
			END_IF;
			IF TX >= TIME_TO_UDINT2(self_act_cycle + self_act_time) THEN
				last := now;
				OUT := FALSE;
				STATUS := BYTE#100;
			END_IF;
		END_IF;
	END_IF;

END_FUNCTION_BLOCK

PROGRAM program0
	VAR
		IN :	BOOL;
		SELF_ACT_CYCLE :	TIME := T#10d;
		SELF_ACT_TIME :	TIME := T#1s;
		OUT :	BOOL;
		STATUS :	BYTE;
		func_block : ACTUATOR_COIL_Block;
	END_VAR
	func_block.IN := IN;
	func_block.SELF_ACT_CYCLE := SELF_ACT_CYCLE;
	func_block.SELF_ACT_TIME := SELF_ACT_TIME ;
	func_block();
	OUT  := func_block.OUT;
	STATUS  := func_block.STATUS;
END_PROGRAM

(* ---- lb_claude_assisted_7111937cfaef_0062.st ---- *)
FUNCTION_BLOCK T_PLC_MS_block
	VAR_OUTPUT
		T_PLC_MS :	UDINT;
	END_VAR

	VAR_EXTERNAL
		PLC_TICKS_PER_SEC :	INT;
		PLC_SYS_TICK_CNT :	DINT;
	END_VAR

	VAR
		debug :	BOOL;(*Debug-Mode ON / OFF*)
		N :	INT;(*Debug-Faktor*)
		Offset :	UDINT;(*Debug-Offset*)
		temp :	DWORD := DWORD#1;(*Debug-Offset*)
		mode :	BOOL;(*modus*)
		faktor :	UDINT;(*Systemtakt-Faktor*)
		init :	BOOL;
		v_plc_ticks_per_sec :	UDINT;
		base :	UDINT := UDINT#1000;
	END_VAR

	IF init = FALSE THEN
		v_plc_ticks_per_sec := INT_TO_UDINT(PLC_TICKS_PER_SEC);
		IF v_plc_ticks_per_sec = UDINT#1024 THEN
			faktor := UDINT#1;
			mode := FALSE;
		ELSIF v_plc_ticks_per_sec > UDINT#0 THEN
			IF v_plc_ticks_per_sec <= base THEN
				faktor := base / v_plc_ticks_per_sec;
				mode := FALSE;
			ELSE
				faktor := v_plc_ticks_per_sec / base;
				mode := TRUE;
			END_IF;
		ELSE
			faktor := UDINT#1;
		END_IF;
		init := TRUE;
	END_IF;

	IF mode THEN
		T_PLC_MS := DINT_TO_UDINT(PLC_SYS_TICK_CNT) / faktor;
	ELSE
		IF init = FALSE THEN
		    T_PLC_MS := DINT_TO_UDINT(PLC_SYS_TICK_CNT) / faktor;
		ELSE
		    T_PLC_MS := DINT_TO_UDINT(PLC_SYS_TICK_CNT) * faktor;
		END_IF;
	END_IF;

	IF debug THEN
		T_PLC_MS := (DWORD_TO_UDINT(SHL(UDINT_TO_DWORD(T_PLC_MS),N) OR SHL(temp,N)) - UDINT#1) + Offset;
	END_IF;
END_FUNCTION_BLOCK

FUNCTION _WORD_TO_DINT:DINT
	VAR_INPUT
		IN :	WORD;
	END_VAR
	_WORD_TO_DINT := UINT_TO_DINT(WORD_TO_UINT(IN));
END_FUNCTION

FUNCTION TIME_TO_UDINT2:UDINT
	VAR_INPUT
		X :	TIME;
	END_VAR

	TIME_TO_UDINT2 := DINT_TO_UDINT(TIME_TO_DINT(X));
END_FUNCTION

FUNCTION_BLOCK _RMP_W

	VAR_INPUT
		DIR :	BOOL;
		E :	BOOL := TRUE;
		TR :	TIME;
	END_VAR

	VAR_IN_OUT
		RMP :	WORD;
	END_VAR

	VAR
		T_PLC_MS :	T_PLC_MS_block;
		tx :	UDINT;
		tl :	UDINT;
		ptesss :	DINT;
		init :	BOOL;
		last_dir :	BOOL;
	END_VAR

	T_PLC_MS();
	tx := T_PLC_MS.T_PLC_MS;
	IF E AND init THEN
		(* we need to set tl = tx when direction changes *)
		IF dir XOR last_dir THEN
			tl := tx;
			last_dir := dir;
		END_IF;
		(* check_elapsed time and calculate only if necessary *)
		IF tr > t#0s THEN
			ptesss := DWORD_TO_DINT(UDINT_TO_DWORD(DWORD_TO_UDINT(SHL(UDINT_TO_DWORD(tx-tl), 16)) / TIME_TO_UDINT2(TR)));
		ELSE
			ptesss := DINT#65535;
		END_IF;
		IF ptesss > DINT#0 THEN
			(* perform the ptesss on the ramp *)
			tl := tx;
			(* calculate the ptesss response *)
			IF NOT dir THEN ptesss := - ptesss; END_IF;
			rmp := DINT_TO_WORD(LIMIT(DINT#0, _WORD_TO_DINT(rmp) + ptesss, DINT#65535));
		END_IF;
	ELSE
		tl := tx;
		init := TRUE;
	END_IF;
END_FUNCTION_BLOCK

FUNCTION_BLOCK RMP_W

	VAR_INPUT
		SET :	BOOL;
		PT :	TIME;
		E :	BOOL := TRUE;
		UP :	BOOL := TRUE;
		RST :	BOOL;
	END_VAR

	VAR_OUTPUT
		OUT :	WORD;
		BUSY :	BOOL;
		HIGH :	BOOL;
		LOW :	BOOL;
	END_VAR

	VAR
		rmp :	_RMP_W;
	END_VAR

	rmp(dir := UP, E := E, TR := PT, rmp := out);
	out := rmp.RMP;

	IF RST THEN
		out := WORD#0;
	ELSIF SET THEN
		out := WORD#65535;
	END_IF;

	low := out = WORD#0;
	high := out = WORD#65535;
	busy := NOT (low OR high) AND E;

END_FUNCTION_BLOCK

PROGRAM program0
  VAR
		SET :	BOOL;
		PT  :	TIME;
		E   :	BOOL;
		UP  :	BOOL ;
		RST :	BOOL;

		OUT  :	WORD;
		BUSY :	BOOL;
		HIGH :	BOOL;
		LOW  :	BOOL;

	func_block : RMP_W;
  END_VAR
	func_block.SET:=SET;
	func_block.PT :=PT ;
	func_block.E  :=E ;
	func_block.UP :=UP ;
	func_block.RST:=RST;
	func_block();
	OUT  := func_block.OUT ;
	BUSY := func_block.BUSY;
	HIGH := func_block.HIGH;
	LOW  := func_block.LOW ;

END_PROGRAM

CONFIGURATION Config0
	VAR_GLOBAL
		PLC_TICKS_PER_SEC :	INT;
		PLC_SYS_TICK_CNT :	DINT;
	END_VAR
  	RESOURCE Res0 ON PLC
    	TASK task0(INTERVAL := T#20ms,PRIORITY := 0);
    	PROGRAM instance0 WITH task0 : program0;
  	END_RESOURCE
END_CONFIGURATION

(* ---- lb_claude_assisted_71a1796c3619_0024.st ---- *)
FUNCTION UDINT_TO_TIME2:TIME

	VAR_INPUT
		IN :	UDINT;
	END_VAR

	UDINT_TO_TIME2 := DINT_TO_TIME(UDINT_TO_DINT(IN));

END_FUNCTION

FUNCTION_BLOCK T_PLC_MS_block
	VAR_OUTPUT
		T_PLC_MS :	UDINT;
	END_VAR

	VAR_EXTERNAL
		PLC_TICKS_PER_SEC :	INT;
		PLC_SYS_TICK_CNT :	DINT;
	END_VAR

	VAR
		debug :	BOOL;(*Debug-Mode ON / OFF*)
		N :	INT;(*Debug-Faktor*)
		Offset :	UDINT;(*Debug-Offset*)
		temp :	DWORD := DWORD#1;(*Debug-Offset*)
		mode :	BOOL;(*modus*)
		faktor :	UDINT;(*Systemtakt-Faktor*)
		init :	BOOL;
		v_plc_ticks_per_sec :	UDINT;
		base :	UDINT := UDINT#1000;
	END_VAR

	IF init = FALSE THEN
		v_plc_ticks_per_sec := INT_TO_UDINT(PLC_TICKS_PER_SEC);
		IF v_plc_ticks_per_sec = UDINT#1024 THEN
			faktor := UDINT#1;
			mode := FALSE;
		ELSIF v_plc_ticks_per_sec > UDINT#0 THEN
			IF v_plc_ticks_per_sec <= base THEN
				faktor := base / v_plc_ticks_per_sec;
				mode := FALSE;
			ELSE
				faktor := v_plc_ticks_per_sec / base;
				mode := TRUE;
			END_IF;
		ELSE
			faktor := UDINT#1;
		END_IF;
		init := TRUE;
	END_IF;

	IF mode THEN
		IF mode THEN
		    T_PLC_MS := DINT_TO_UDINT(PLC_SYS_TICK_CNT) * faktor;
		ELSE
		    T_PLC_MS := DINT_TO_UDINT(PLC_SYS_TICK_CNT) / faktor;
		END_IF;
	ELSE
		T_PLC_MS := DINT_TO_UDINT(PLC_SYS_TICK_CNT) * faktor;
	END_IF;

	IF debug THEN
		T_PLC_MS := (DWORD_TO_UDINT(SHL(UDINT_TO_DWORD(T_PLC_MS),N) OR SHL(temp,N)) - UDINT#1) + Offset;
	END_IF;

END_FUNCTION_BLOCK

FUNCTION MODR : REAL
  VAR_INPUT
    IN : REAL;
    DIVI : REAL;
  END_VAR

  IF divi = 0.0 THEN
  	MODR := 0.0;
  ELSE
  	MODR := in - DINT_TO_REAL(FLOOR2(in / divi)) * divi;
  END_IF;
END_FUNCTION

FUNCTION FLOOR2 : DINT
  VAR_INPUT
    x : REAL;
  END_VAR

  FLOOR2 := REAL_TO_DINT(X);
  IF DINT_TO_REAL(FLOOR2) > X THEN
  	FLOOR2 := FLOOR2 - DINT#1;
  END_IF;
END_FUNCTION

FUNCTION _REAL_TO_DWORD: DWORD

  VAR_INPUT
    X :	REAL;
  END_VAR

  IF REAL_TO_DWORD(0.5) = DWORD#1 THEN
    _REAL_TO_DWORD := REAL_TO_DWORD(x);
  ELSIF X > 0.0 THEN
    _REAL_TO_DWORD := REAL_TO_DWORD(x+0.5);
  ELSIF X < 0.0 THEN
    _REAL_TO_DWORD := REAL_TO_DWORD(x-0.5);
  ELSE
    _REAL_TO_DWORD := DWORD#0;
  END_IF;
END_FUNCTION

FUNCTION _DWORD_TO_REAL:REAL
	VAR_INPUT
		IN :	DWORD;
	END_VAR

	_DWORD_TO_REAL := UDINT_TO_REAL(DWORD_TO_UDINT(IN));

END_FUNCTION

FUNCTION MULTIME:TIME
	VAR_INPUT
		T :	TIME;
		M :	REAL;
	END_VAR

	multime := DWORD_TO_TIME(_REAL_TO_DWORD(_DWORD_TO_REAL(TIME_TO_DWORD(t))*M));
END_FUNCTION

FUNCTION_BLOCK GEN_SQR_Block

	VAR_INPUT
		PT :	TIME;
		AM :	REAL := REAL#1.0;
		OS :	REAL;
		DC :	REAL := REAL#0.5;
		DL :	REAL;
	END_VAR

	VAR_OUTPUT
		Q :	BOOL;
		Out :	REAL;
	END_VAR

	VAR
		tx :	TIME;
		last :	TIME;
		init :	BOOL;
		T_PLC_MS :	T_PLC_MS_Block;
	END_VAR

	IF dc = 0.0 THEN
		out := -am * 0.5 + os;
		Q := FALSE;
		RETURN;
	ELSIF dc = 1.0 THEN
		out := am * 0.5 + os;
		Q := TRUE;
		RETURN;
	END_IF;

	T_PLC_MS();
	tx:= UDINT_TO_TIME(T_PLC_MS.T_PLC_MS) - last;
	DL := modR(dl,1.0);
	IF dl < 0.0 THEN dl := 1.0 - dl; END_IF;
	dc := modR(dc,1.0);
	IF dc < 0.0 THEN dc := 1.0 - dc; END_IF;

	IF NOT init THEN
		init := TRUE;
		last := tx;
		tx := t#0s;
	END_IF;

	IF tx >= pt THEN
		last := last + pt;
		tx := tx - pt;
	END_IF;

	IF multime(pt, dl + dc) >= pt THEN
		IF tx >= multime(pt, dl + dc - 1.0) THEN
			out := -am * 0.5 + os;
			Q := FALSE;
		END_IF;
		IF tx >= multime(pt, dl) THEN
			out := am * 0.5 + os;
			Q := TRUE;
		END_IF;
	ELSE
		IF tx >= multime(pt, dl) THEN
			out := am * 0.5 + os;
			Q := TRUE;
		END_IF;
		IF tx >= multime(pt, dl + dc) THEN
			out := -am * 0.5 +os;
			Q := FALSE;
		END_IF;
	END_IF;

END_FUNCTION_BLOCK

PROGRAM program0
  VAR
	PT :	TIME;
	AM :	REAL := REAL#1.0;
	OS :	REAL;
	DC :	REAL := REAL#0.5;
	DL :	REAL;
	Q :	BOOL;
	Out :	REAL;
	func_block : GEN_SQR_Block;
  END_VAR
	func_block.PT  :=PT;
	func_block.AM  :=AM;
	func_block.OS  :=OS;
	func_block.DC  :=DC;
	func_block.DL  :=DL;
	func_block();
	Q := func_block.Q;
	OUT := func_block.OUT;
END_PROGRAM

CONFIGURATION Config0
	VAR_GLOBAL
		PLC_TICKS_PER_SEC :	INT;
		PLC_SYS_TICK_CNT :	DINT;
	END_VAR
	RESOURCE Res0 ON PLC
		TASK task0(INTERVAL := T#20ms,PRIORITY := 0);
		PROGRAM instance0 WITH task0 : program0;
	END_RESOURCE
END_CONFIGURATION

(* ---- lb_claude_assisted_747adee92625_0024.st ---- *)
TYPE
  LOGLEVEL : (CRITICAL, WARNING, INFO, DEBUG) := INFO;
END_TYPE

FUNCTION_BLOCK LOGGER
  VAR_INPUT
    TRIG : BOOL;
    MSG : STRING;
    LEVEL : LOGLEVEL := INFO;
  END_VAR
  VAR
    TRIG0 : BOOL;
  END_VAR

  IF TRIG AND NOT TRIG0 THEN
  {{
   LogMessage(GetFbVar(LEVEL),(char*)GetFbVar(MSG, .body),GetFbVar(MSG, .len));
  }}
  END_IF;
  TRIG0:=TRIG;
END_FUNCTION_BLOCK

FUNCTION_BLOCK python_eval
  VAR_INPUT
    TRIG : BOOL;
    CODE : STRING;
  END_VAR
  VAR_OUTPUT
    ACK : BOOL;
    RESULT : STRING;
  END_VAR
  VAR
    STATE : DWORD;
    BUFFER : STRING;
    PREBUFFER : STRING;
    TRIGM1 : BOOL;
    TRIGGED : BOOL;
  END_VAR

  {extern void __PythonEvalFB(int, PYTHON_EVAL*);__PythonEvalFB(0, data__);}
END_FUNCTION_BLOCK

FUNCTION_BLOCK python_poll
  VAR_INPUT
    TRIG : BOOL;
    CODE : STRING;
  END_VAR
  VAR_OUTPUT
    ACK : BOOL;
    RESULT : STRING;
  END_VAR
  VAR
    STATE : DWORD;
    BUFFER : STRING;
    PREBUFFER : STRING;
    TRIGM1 : BOOL;
    TRIGGED : BOOL;
  END_VAR

  {extern void __PythonEvalFB(int, PYTHON_EVAL*);__PythonEvalFB(1,(PYTHON_EVAL*)(void*)data__);}
END_FUNCTION_BLOCK

FUNCTION_BLOCK python_gear
  VAR_INPUT
    N : UINT;
    TRIG : BOOL;
    CODE : STRING;
  END_VAR
  VAR_OUTPUT
    ACK : BOOL;
    RESULT : STRING;
  END_VAR
  VAR
    py_eval : python_eval;
    COUNTER : UINT;
    ADD10_OUT : UINT;
    EQ13_OUT : BOOL;
    SEL15_OUT : UINT;
    AND7_OUT : BOOL;
  END_VAR

  ADD10_OUT := ADD(COUNTER, 1);
  EQ13_OUT := EQ(N, ADD10_OUT);
  SEL15_OUT := SEL(EQ13_OUT, ADD10_OUT, 0);
  COUNTER := SEL15_OUT;
  AND7_OUT := AND(EQ13_OUT, TRIG);
  py_eval(TRIG := AND7_OUT, CODE := CODE);
  ACK := py_eval.ACK;
  RESULT := py_eval.RESULT;
END_FUNCTION_BLOCK

FUNCTION_BLOCK GetBoolString
  VAR_INPUT
    VALUE : BOOL;
  END_VAR
  VAR_OUTPUT
    CODE : STRING;
  END_VAR

  IF VALUE THEN
    CODE := 'True';
  ELSE
    CODE := 'False';
  END_IF;
END_FUNCTION_BLOCK

FUNCTION_BLOCK Button
  VAR
    ID : STRING;
  END_VAR
  VAR_INPUT
    back_id : STRING;
    sele_id : STRING;
    toggle : BOOL;
    set_state : BOOL;
    state_in : BOOL;
  END_VAR
  VAR_OUTPUT
    state_out : BOOL;
  END_VAR
  VAR
    init_Command : python_eval;
    GetButtonState : GetBoolString;
    setstate_Command : python_eval;
    getstate_Command : python_poll;
    GetButtonToggle : GetBoolString;
    CONCAT2_OUT : STRING;
    CONCAT22_OUT : STRING;
    STRING_TO_INT25_OUT : INT;
    INT_TO_BOOL26_OUT : BOOL;
    AND31_OUT : BOOL;
    CONCAT7_OUT : STRING;
  END_VAR

  GetButtonToggle(VALUE := toggle);
  CONCAT2_OUT := CONCAT('createSVGUIControl("button",back_id="', back_id, '",sele_id="', sele_id, '",toggle=', GetButtonToggle.CODE, ',active=True)');
  init_Command(TRIG := BOOL#1, CODE := CONCAT2_OUT);
  ID := init_Command.RESULT;
  CONCAT22_OUT := CONCAT('int(getAttr(', ID, ',"state",False))');
  getstate_Command(TRIG := init_Command.ACK, CODE := CONCAT22_OUT);
  STRING_TO_INT25_OUT := STRING_TO_INT(getstate_Command.RESULT);
  INT_TO_BOOL26_OUT := INT_TO_BOOL(STRING_TO_INT25_OUT);
  state_out := INT_TO_BOOL26_OUT;
  AND31_OUT := AND(init_Command.ACK, set_state);
  GetButtonState(VALUE := state_in);
  CONCAT7_OUT := CONCAT('setAttr(', ID, ',"state",', GetButtonState.CODE, ')');
  setstate_Command(TRIG := AND31_OUT, CODE := CONCAT7_OUT);
END_FUNCTION_BLOCK

FUNCTION_BLOCK Led
  VAR
    ID : STRING;
  END_VAR
  VAR_INPUT
    back_id : STRING;
    sele_id : STRING;
    state_in : BOOL;
  END_VAR
  VAR
    init_Command : python_eval;
    setstate_Command : python_poll;
    GetLedState : GetBoolString;
    CONCAT2_OUT : STRING;
    CONCAT7_OUT : STRING;
  END_VAR

  CONCAT2_OUT := CONCAT('createSVGUIControl("button",back_id="', back_id, '",sele_id="', sele_id, '",toggle=True,active=False)');
  init_Command(TRIG := BOOL#1, CODE := CONCAT2_OUT);
  ID := init_Command.RESULT;
  GetLedState(VALUE := state_in);
  CONCAT7_OUT := CONCAT('setAttr(', ID, ',"state",', GetLedState.CODE, ')');
  setstate_Command(TRIG := init_Command.ACK, CODE := CONCAT7_OUT);
END_FUNCTION_BLOCK

FUNCTION_BLOCK TextCtrl
  VAR
    ID : STRING;
  END_VAR
  VAR_INPUT
    back_id : STRING;
    set_text : BOOL;
    text : STRING;
  END_VAR
  VAR
    SVGUI_TEXTCTRL : python_eval;
    setstate_Command : python_eval;
    CONCAT1_OUT : STRING;
    AND31_OUT : BOOL;
    CONCAT12_OUT : STRING;
  END_VAR

  CONCAT1_OUT := CONCAT('createSVGUIControl("textControl", back_id="', back_id, '")');
  SVGUI_TEXTCTRL(TRIG := BOOL#1, CODE := CONCAT1_OUT);
  ID := SVGUI_TEXTCTRL.RESULT;
  AND31_OUT := AND(SVGUI_TEXTCTRL.ACK, set_text);
  CONCAT12_OUT := CONCAT('setAttr(', ID, ',"text","', text, '")');
  setstate_Command(TRIG := AND31_OUT, CODE := CONCAT12_OUT);
END_FUNCTION_BLOCK

FUNCTION_BLOCK CounterSFC
  VAR_INPUT
    Reset : BOOL;
  END_VAR
  VAR_OUTPUT
    OUT : INT;
  END_VAR
  VAR
    Cnt : INT;
  END_VAR
  VAR_EXTERNAL CONSTANT
    ResetCounterValue : INT;
  END_VAR

  INITIAL_STEP Start:
  END_STEP

  TRANSITION FROM Start TO ResetCounter
    := Reset;
  END_TRANSITION

  STEP ResetCounter:
    RESETCOUNTER_INLINE1(N);
    RESETCOUNTER_INLINE2(N);
  END_STEP

  ACTION RESETCOUNTER_INLINE1:
    Cnt := ResetCounterValue;
  END_ACTION

  ACTION RESETCOUNTER_INLINE2:
    OUT := Cnt;
  END_ACTION

  TRANSITION FROM ResetCounter TO Start
    := NOT Reset;
  END_TRANSITION

  TRANSITION FROM Start TO Count
    := NOT Reset;
  END_TRANSITION

  STEP Count:
    COUNT_INLINE3(N);
    COUNT_INLINE4(N);
  END_STEP

  ACTION COUNT_INLINE3:
    Cnt := Cnt + 1;
  END_ACTION

  ACTION COUNT_INLINE4:
    OUT := Cnt;
  END_ACTION

  TRANSITION FROM Count TO Start
    := Reset;
  END_TRANSITION

END_FUNCTION_BLOCK

FUNCTION_BLOCK CounterFBD
  VAR_INPUT
    Reset : BOOL;
  END_VAR
  VAR_OUTPUT
    OUT : INT;
  END_VAR
  VAR
    Cnt : INT;
  END_VAR
  VAR_EXTERNAL CONSTANT
    ResetCounterValue : INT;
  END_VAR
  VAR
    ADD4_OUT : INT;
    SEL7_OUT : INT;
  END_VAR

  ADD4_OUT := ADD(1, Cnt);
  SEL7_OUT := SEL(Reset, ADD4_OUT, ResetCounterValue);
  Cnt := SEL7_OUT;
  OUT := Cnt;
END_FUNCTION_BLOCK

FUNCTION_BLOCK CounterIL
  VAR
    Cnt : INT;
  END_VAR
  VAR_INPUT
    Reset : BOOL;
  END_VAR
  VAR_OUTPUT
    OUT : INT;
  END_VAR
  VAR_EXTERNAL CONSTANT
    ResetCounterValue : INT;
  END_VAR

  LD Reset
  JMPC ResetCnt

  (* increment counter *)
  LD Cnt
  ADD 1
  JMP QuitFb

  ResetCnt:
  (* reset counter *)
  LD ResetCounterValue

  QuitFb:
  (* save results *)
  ST Cnt
  ST Out
END_FUNCTION_BLOCK

FUNCTION_BLOCK CounterST
  VAR_INPUT
    Reset : BOOL;
  END_VAR
  VAR
    Cnt : INT;
  END_VAR
  VAR_OUTPUT
    OUT : INT;
  END_VAR
  VAR_EXTERNAL CONSTANT
    ResetCounterValue : INT;
  END_VAR

  IF Reset THEN
    IF Reset THEN
        Cnt := Cnt + 1;
    ELSE
        Cnt := ResetCounterValue;
    END_IF;
  ELSE
    Cnt := Cnt + 1;
  END_IF;

  Out := Cnt;
END_FUNCTION_BLOCK

FUNCTION_BLOCK CounterLD
  VAR_INPUT
    Reset : BOOL;
  END_VAR
  VAR_OUTPUT
    Out : INT;
  END_VAR
  VAR
    Cnt : INT;
  END_VAR
  VAR_EXTERNAL CONSTANT
    ResetCounterValue : INT;
  END_VAR
  VAR
    ADD4_OUT : INT;
    SEL7_OUT : INT;
  END_VAR

  ADD4_OUT := ADD(1, Cnt);
  SEL7_OUT := SEL(Reset, ADD4_OUT, ResetCounterValue);
  Cnt := SEL7_OUT;
  Out := Cnt;
END_FUNCTION_BLOCK

PROGRAM plc_prg
  VAR_INPUT
    Reset : BOOL;
  END_VAR
  VAR_OUTPUT
    Cnt1 : INT;
    Cnt2 : INT;
    Cnt3 : INT;
    Cnt4 : INT;
    Cnt5 : INT;
  END_VAR
  VAR
    CounterST0 : CounterST;
    CounterFBD0 : CounterFBD;
    CounterSFC0 : CounterSFC;
    CounterIL0 : CounterIL;
    CounterLD0 : CounterLD;
  END_VAR

  CounterST0(Reset := Reset);
  Cnt1 := CounterST0.OUT;
  CounterFBD0(Reset := Reset);
  Cnt2 := CounterFBD0.OUT;
  CounterSFC0(Reset := Reset);
  Cnt3 := CounterSFC0.OUT;
  CounterIL0(Reset := Reset);
  Cnt4 := CounterIL0.OUT;
  CounterLD0(Reset := Reset);
  Cnt5 := CounterLD0.Out;
END_PROGRAM

CONFIGURATION config
  VAR_GLOBAL CONSTANT
    ResetCounterValue : INT := 17;
  END_VAR

  RESOURCE resource1 ON PLC
    TASK plc_task(INTERVAL := T#100ms,PRIORITY := 1);
    PROGRAM plc_task_instance WITH plc_task : plc_prg;
  END_RESOURCE
END_CONFIGURATION

(* ---- lb_claude_assisted_7a3faffe2dcc_0005.st ---- *)
(*
This code implements a randomly grown symbolic expression:

xor(xor((IN16 | IN26) & ((((xor(xor(!(xor(xor(IN38 | (!(IN38)), !(!(IN8))), !(xor(xor(IN44, IN37), IN27)))), (((!(IN1)) & (IN27 | IN45)) | (IN40 & (IN38 & IN27))) & IN36), ((!(!(IN43))) | ((xor(xor(IN16, IN18), IN25)) & (IN45 & IN43))) & (((!(IN16)) | (IN31 & IN9)) & (xor(xor(IN8, IN40), IN38 | IN17))))) & (xor(xor(((!(IN27)) & ((!(IN1)) | (IN35 & IN28))) | ((!(!(IN15))) & IN32), (((IN48 & IN5) | (IN10 | true)) | true) | (xor(xor(false, !(xor(xor(IN43, IN3), IN44))), xor(xor(xor(xor(IN49, IN34), IN16), IN12 | IN26), IN6)))), (IN39 & (xor(xor(IN46 & IN10, IN22 | IN11), xor(xor(IN46, IN12), true)))) | IN28))) | (!((xor(xor(xor(xor((IN45 | IN44) | (IN15 | IN13), (!(IN36)) | (IN45 | IN39)), !(IN9 & IN49)), (xor(xor(xor(xor(IN4, IN37), IN21), xor(xor(IN9, IN19), IN3)), IN30 & IN16)) | (!(xor(xor(IN25, IN45), IN33)))), ((IN40 & IN16) | (!(IN39))) | ((xor(xor(IN25, IN35), IN21)) & (IN30 & IN29)))) | (xor(xor(IN16, (!(IN5 & IN15)) | (!(!(IN18)))), IN49))))) & (IN39 | (!(((IN38 & IN11) & (!((!(IN25)) | (!(IN2))))) | IN25)))), IN25), IN6 & ((!(xor(xor(!(xor(xor(xor(xor((xor(xor(IN45, IN32), IN43)) & (IN9 | IN44), false), xor(xor(IN13 | IN25, IN9 & IN14), IN48 | IN42)), !((!(IN11)) & (!(IN27)))), (!(IN25)) | (!(!(IN48))))), (!(IN15)) | (xor(xor(xor(xor((xor(xor(IN48, false), IN4)) & (xor(xor(IN34, IN46), IN33)), !(xor(xor(IN7, IN46), IN31))), xor(xor(!(IN13), false & IN43), xor(xor(IN13, IN36), IN26))), ((false | IN10) | (IN24 | IN15)) & IN38), IN14 | (xor(xor(IN50, xor(xor(IN3, IN1), IN14)), !(IN43)))))), !((xor(xor(!(xor(xor(IN23, false), IN25)), xor(xor(xor(xor(IN21, IN7), IN18), IN32 | IN34), xor(xor(IN28, IN2), IN43))), IN35)) | (((!(IN47)) & (IN50 | IN28)) | (xor(xor(IN45 | IN1, IN16 & IN45), IN29))))))) & (xor(xor(!(xor(xor(xor(xor(IN32, xor(xor(!(IN42 & IN4), IN22), IN42 & (!(IN46)))), xor(xor(IN6, (!(IN37)) | (IN11 & IN40)), (!(IN50)) | (false & IN45))), !((IN20 | (!(IN44))) & IN32)), !(((xor(xor(IN19, IN36), IN22)) | (IN38 & IN45)) & (!(!(IN35)))))), xor(xor(!(IN34), (!(IN3)) | IN50), !((xor(xor((IN16 | IN18) & IN41, xor(xor(IN50, xor(xor(IN2, IN44), IN23)), xor(xor(IN8, IN43), IN19))), xor(xor(IN11 | IN29, !(IN44)), !(IN27)))) | IN45))), (!((!(IN30 | (xor(xor(IN45, IN14), IN20)))) & (xor(xor(!(IN18), (IN13 | false) & (IN8 & IN46)), IN28)))) | IN20))))

*)

FUNCTION_BLOCK F_CollectInput
  VAR_IN_OUT
      Data : ARRAY[1..50] OF BOOL;
  END_VAR
  VAR_INPUT
      TICK  : BOOL := 0;
      IN1   : BOOL := 0;
      IN2   : BOOL := 0;
      IN3   : BOOL := 0;
      IN4   : BOOL := 0;
      IN5   : BOOL := 0;
      RESET : BOOL := FALSE;
  END_VAR
  VAR_OUTPUT
      Finished : BOOL;
  END_VAR
  VAR
      j    : USINT := 1;
      tock : BOOL  := 0;
  END_VAR
  IF NOT RESET AND tock = NOT TICK THEN
      Data[j]   := IN1;
      Data[j+1] := IN2;
      Data[j+2] := IN3;
      Data[j+3] := IN4;
      Data[j+4] := IN5;
      j := j + 5;
      tock := TICK;
  ELSE
      j := 1;
      tock := 0;
  END_IF;
  Finished := (j > 50);
END_FUNCTION_BLOCK

PROGRAM Boiler
  VAR
    Data  : ARRAY[1..50] OF BOOL;
    Ready : BOOL;
    CollectInput : F_CollectInput;
  END_VAR
  VAR
    TICK     AT %IX1.0 : BOOL;
    IN1      AT %IX0.3 : BOOL;
    IN2      AT %IX0.4 : BOOL;
    IN3      AT %IX0.5 : BOOL;
    IN4      AT %IX0.6 : BOOL;
    IN5      AT %IX0.7 : BOOL;
    OutReady AT %QX0.0 : BOOL := FALSE;
    FeedNext AT %QX0.1 : BOOL := FALSE;
    Out      AT %QX0.2 : BOOL;
  END_VAR
  CollectInput(TICK:=TICK, IN1:=IN1, IN2:=IN2, IN3:=IN3, IN4:=IN4, IN5:=IN5);
  Ready := CollectInput.Finished;
  FeedNext := 1;
  IF Ready THEN
    Out := ((((Data[16] OR Data[26]) AND ((((((NOT (((Data[38] OR (NOT Data[38])) XOR (NOT (NOT Data[8]))) XOR (NOT ((Data[44] XOR Data[37]) XOR Data[27])))) XOR ((((NOT Data[1]) AND (Data[27] OR Data[45])) OR (Data[40] AND (Data[38] AND Data[27]))) AND Data[36])) XOR (((NOT (NOT Data[43])) OR (((Data[16] XOR Data[18]) XOR Data[25]) AND (Data[45] AND Data[43]))) AND (((NOT Data[16]) OR (Data[31] AND Data[9])) AND ((Data[8] XOR Data[40]) XOR (Data[38] OR Data[17]))))) AND (((((NOT Data[27]) AND ((NOT Data[1]) OR (Data[35] AND Data[28]))) OR ((NOT (NOT Data[15])) AND Data[32])) XOR ((((Data[48] AND Data[5]) OR (Data[10] OR TRUE)) OR TRUE) OR ((FALSE XOR (NOT ((Data[43] XOR Data[3]) XOR Data[44]))) XOR ((((Data[49] XOR Data[34]) XOR Data[16]) XOR (Data[12] OR Data[26])) XOR Data[6])))) XOR ((Data[39] AND (((Data[46] AND Data[10]) XOR (Data[22] OR Data[11])) XOR ((Data[46] XOR Data[12]) XOR TRUE))) OR Data[28]))) OR (NOT (((((((Data[45] OR Data[44]) OR (Data[15] OR Data[13])) XOR ((NOT Data[36]) OR (Data[45] OR Data[39]))) XOR (NOT (Data[9] AND Data[49]))) XOR (((((Data[4] XOR Data[37]) XOR Data[21]) XOR ((Data[9] XOR Data[19]) XOR Data[3])) XOR (Data[30] AND Data[16])) OR (NOT ((Data[25] XOR Data[45]) XOR Data[33])))) XOR (((Data[40] AND Data[16]) OR (NOT Data[39])) OR (((Data[25] XOR Data[35]) XOR Data[21]) AND (Data[30] AND Data[29])))) OR ((Data[16] XOR ((NOT (Data[5] AND Data[15])) OR (NOT (NOT Data[18])))) XOR Data[49])))) AND (Data[39] OR (NOT (((Data[38] AND Data[11]) AND (NOT ((NOT Data[25]) OR (NOT Data[2])))) OR Data[25]))))) XOR Data[25]) XOR (Data[6] AND ((NOT (((NOT (((((((Data[45] XOR Data[32]) XOR Data[43]) AND (Data[9] OR Data[44])) XOR FALSE) XOR (((Data[13] OR Data[25]) XOR (Data[9] AND Data[14])) XOR (Data[48] OR Data[42]))) XOR (NOT ((NOT Data[11]) AND (NOT Data[27])))) XOR ((NOT Data[25]) OR (NOT (NOT Data[48]))))) XOR ((NOT Data[15]) OR (((((((Data[48] XOR FALSE) XOR Data[4]) AND ((Data[34] XOR Data[46]) XOR Data[33])) XOR (NOT ((Data[7] XOR Data[46]) XOR Data[31]))) XOR (((NOT Data[13]) XOR (FALSE AND Data[43])) XOR ((Data[13] XOR Data[36]) XOR Data[26]))) XOR (((FALSE OR Data[10]) OR (Data[24] OR Data[15])) AND Data[38])) XOR (Data[14] OR ((Data[50] XOR ((Data[3] XOR Data[1]) XOR Data[14])) XOR (NOT Data[43])))))) XOR (NOT ((((NOT ((Data[23] XOR FALSE) XOR Data[25])) XOR ((((Data[21] XOR Data[7]) XOR Data[18]) XOR (Data[32] OR Data[34])) XOR ((Data[28] XOR Data[2]) XOR Data[43]))) XOR Data[35]) OR (((NOT Data[47]) AND (Data[50] OR Data[28])) OR (((Data[45] OR Data[1]) XOR (Data[16] AND Data[45])) XOR Data[29])))))) AND (((NOT ((((Data[32] XOR (((NOT (Data[42] AND Data[4])) XOR Data[22]) XOR (Data[42] AND (NOT Data[46])))) XOR ((Data[6] XOR ((NOT Data[37]) OR (Data[11] AND Data[40]))) XOR ((NOT Data[50]) OR (FALSE AND Data[45])))) XOR (NOT ((Data[20] OR (NOT Data[44])) AND Data[32]))) XOR (NOT ((((Data[19] XOR Data[36]) XOR Data[22]) OR (Data[38] AND Data[45])) AND (NOT (NOT Data[35])))))) XOR (((NOT Data[34]) XOR ((NOT Data[3]) OR Data[50])) XOR (NOT (((((Data[16] OR Data[18]) AND Data[41]) XOR ((Data[50] XOR ((Data[2] XOR Data[44]) XOR Data[23])) XOR ((Data[8] XOR Data[43]) XOR Data[19]))) XOR (((Data[11] OR Data[29]) XOR (NOT Data[44])) XOR (NOT Data[27]))) OR Data[45])))) XOR ((NOT ((NOT (Data[30] OR ((Data[45] XOR Data[14]) XOR Data[20]))) AND (((NOT Data[18]) XOR ((Data[13] OR FALSE) AND (Data[8] AND Data[46]))) XOR Data[28]))) OR Data[20])))));
    IF Ready THEN
        OutReady := 0;
    ELSE
        OutReady := 1;
    END_IF;
    CollectInput(RESET:=TRUE);
  END_IF;
END_PROGRAM

CONFIGURATION Config0
  RESOURCE Res0 ON PLC
    TASK task0(INTERVAL := T#20ms,PRIORITY := 0);
    PROGRAM instance0 WITH task0 : Boiler;
  END_RESOURCE
END_CONFIGURATION

(* ---- lb_claude_assisted_7aba08e64a94_0066.st ---- *)
FUNCTION_BLOCK T_PLC_MS_block
	VAR_OUTPUT
		T_PLC_MS :	UDINT;
	END_VAR

	VAR
		PLC_TICKS_PER_SEC :	INT;
		PLC_SYS_TICK_CNT :	DINT;
	END_VAR

	VAR
		debug :	BOOL;(*Debug-Mode ON / OFF*)
		N :	INT;(*Debug-Faktor*)
		Offset :	UDINT;(*Debug-Offset*)
		temp :	DWORD := DWORD#1;(*Debug-Offset*)
		MODE :	BOOL;(*modus*)
		faktor :	UDINT;(*Systemtakt-Faktor*)
		init :	BOOL;
		v_plc_ticks_per_sec :	UDINT;
		base :	UDINT := UDINT#1000;
	END_VAR

	IF init = FALSE THEN
		v_plc_ticks_per_sec := INT_TO_UDINT(PLC_TICKS_PER_SEC);
		IF v_plc_ticks_per_sec = UDINT#1024 THEN
			faktor := UDINT#1;
			MODE := FALSE;
		ELSIF v_plc_ticks_per_sec > UDINT#0 THEN
			IF v_plc_ticks_per_sec <= base THEN
				faktor := base / v_plc_ticks_per_sec;
				MODE := FALSE;
			ELSE
				faktor := v_plc_ticks_per_sec / base;
				MODE := TRUE;
			END_IF;
		ELSE
			faktor := UDINT#1;
		END_IF;
		init := TRUE;
	END_IF;

	IF MODE THEN
		T_PLC_MS := DINT_TO_UDINT(PLC_SYS_TICK_CNT) / faktor;
	ELSE
		IF NOT MODE THEN
		    T_PLC_MS := DINT_TO_UDINT(PLC_SYS_TICK_CNT) / faktor;
		ELSE
		    T_PLC_MS := DINT_TO_UDINT(PLC_SYS_TICK_CNT) * faktor;
		END_IF;
	END_IF;

	IF debug THEN
		T_PLC_MS := (DWORD_TO_UDINT(SHL(UDINT_TO_DWORD(T_PLC_MS),N) OR SHL(temp,N)) - UDINT#1) + Offset;
	END_IF;

END_FUNCTION_BLOCK

FUNCTION_BLOCK CLK_PRG
	VAR_INPUT
		PT :	TIME := T#10ms;
	END_VAR

	VAR_OUTPUT
		Q :	BOOL;
	END_VAR

	VAR
		init :	BOOL := FALSE;
		last :	TIME;
		TX :	TIME;
		T_PLC_MS :	T_PLC_MS_block;
	END_VAR

	T_PLC_MS();
	TX:= UDINT_TO_TIME(T_PLC_MS.T_PLC_MS);

	IF NOT init THEN
		init := TRUE;
		last := SUB_TIME(TX, PT);
	END_IF;

	Q := SUB_TIME(TX, last) >= PT;
	IF Q THEN last := TX; END_IF;
END_FUNCTION_BLOCK

FUNCTION _REAL_TO_UDINT:UDINT
  VAR_INPUT
    X :	REAL;
  END_VAR

  IF REAL_TO_UDINT(0.5) = UDINT#1 THEN
    _REAL_TO_UDINT := REAL_TO_UDINT(X);
  ELSIF X > 0.0 THEN
    _REAL_TO_UDINT := REAL_TO_UDINT(X+0.5);
  ELSIF X < 0.0 THEN
    _REAL_TO_UDINT := REAL_TO_UDINT(X-0.5);
  ELSE
    _REAL_TO_UDINT := UDINT#0;
  END_IF;
END_FUNCTION

FUNCTION REAL_TO_TIME2:TIME
	VAR_INPUT
		IN :	REAL;
	END_VAR

	REAL_TO_TIME2 := DINT_TO_TIME(UDINT_TO_DINT(_REAL_TO_UDINT(IN)));
END_FUNCTION

FUNCTION_BLOCK TP_X
	VAR_INPUT
		IN :	BOOL;
		PT :	TIME;
	END_VAR

	VAR_OUTPUT
		Q :	BOOL;
		ET :	TIME;
	END_VAR

	VAR
		edge :	BOOL;
		START :	TIME;
		TX :	TIME;
		T_PLC_MS :	T_PLC_MS_block;
	END_VAR

	T_PLC_MS();
	TX := UDINT_TO_TIME(T_PLC_MS.T_PLC_MS);

	IF IN AND NOT edge THEN
		START := TX;
		Q := PT > t#0ms;
	ELSIF Q THEN
		ET := TX - START;
		IF ET >= PT THEN
			Q := FALSE;
			ET := t#0ms;
		END_IF;
	END_IF;
	edge := IN;

END_FUNCTION_BLOCK

FUNCTION_BLOCK PWM_DC
	VAR_INPUT
		F :	REAL;
		DC :	REAL;
	END_VAR

	VAR_OUTPUT
		Q :	BOOL;
	END_VAR

	VAR
		CLK :	CLK_Prg;
		pulse :	TP_X;
		tmp :	REAL;
	END_VAR

	IF F > 0.0 THEN
		tmp := 1000.0/F;
		CLK(PT := REAL_TO_TIME2(tmp));
		Pulse(IN := CLK.Q, PT := REAL_TO_TIME2(tmp*DC));
		Q := pulse.Q;
	END_IF;
END_FUNCTION_BLOCK

PROGRAM program0
  VAR
	F  :	REAL;
	DC :	REAL;

	Q :	BOOL;

	func_block : PWM_DC;
  END_VAR
	func_block.F     :=F     ;
	func_block.DC    :=DC    ;
	func_block();
	Q := func_block.Q;
END_PROGRAM

(* ---- lb_claude_assisted_7de25bc7b92f_0050.st ---- *)
FUNCTION _REAL_TO_DWORD: DWORD

  VAR_INPUT
    X :	REAL;
  END_VAR

  IF REAL_TO_DWORD(0.5) = DWORD#1 THEN
    _REAL_TO_DWORD := REAL_TO_DWORD(x);
  ELSIF X > 0.0 THEN
    _REAL_TO_DWORD := REAL_TO_DWORD(x+0.5);
  ELSIF X < 0.0 THEN
    _REAL_TO_DWORD := REAL_TO_DWORD(x-0.5);
  ELSE
    _REAL_TO_DWORD := DWORD#0;
  END_IF;
END_FUNCTION

FUNCTION _DWORD_TO_REAL:REAL
	VAR_INPUT
		IN :	DWORD;
	END_VAR

	_DWORD_TO_REAL := UDINT_TO_REAL(DWORD_TO_UDINT(IN));

END_FUNCTION

FUNCTION MULTIME:TIME
	VAR_INPUT
		T :	TIME;
		M :	REAL;
	END_VAR

	multime := DWORD_TO_TIME(_REAL_TO_DWORD(_DWORD_TO_REAL(TIME_TO_DWORD(t))*M));
END_FUNCTION

FUNCTION UDINT_TO_TIME2:TIME

	VAR_INPUT
		IN :	UDINT;
	END_VAR

	UDINT_TO_TIME2 := DINT_TO_TIME(UDINT_TO_DINT(IN));

END_FUNCTION

FUNCTION_BLOCK T_PLC_MS_block
	VAR_OUTPUT
		T_PLC_MS :	UDINT;
	END_VAR

	VAR_EXTERNAL
		PLC_TICKS_PER_SEC :	INT;
		PLC_SYS_TICK_CNT :	DINT;
	END_VAR

	VAR
		debug :	BOOL;(*Debug-Mode ON / OFF*)
		N :	INT;(*Debug-Faktor*)
		Offset :	UDINT;(*Debug-Offset*)
		temp :	DWORD := DWORD#1;(*Debug-Offset*)
		mode :	BOOL;(*modus*)
		faktor :	UDINT;(*Systemtakt-Faktor*)
		init :	BOOL;
		v_plc_ticks_per_sec :	UDINT;
		base :	UDINT := UDINT#1000;
	END_VAR

	IF init = FALSE THEN
		v_plc_ticks_per_sec := INT_TO_UDINT(PLC_TICKS_PER_SEC);
		IF v_plc_ticks_per_sec = UDINT#1024 THEN
			faktor := UDINT#1;
			mode := FALSE;
		ELSIF v_plc_ticks_per_sec > UDINT#0 THEN
			IF v_plc_ticks_per_sec <= base THEN
				faktor := base / v_plc_ticks_per_sec;
				mode := FALSE;
			ELSE
				faktor := v_plc_ticks_per_sec / base;
				mode := TRUE;
			END_IF;
		ELSE
			faktor := UDINT#1;
		END_IF;
		init := TRUE;
	END_IF;

	IF mode THEN
		T_PLC_MS := DINT_TO_UDINT(PLC_SYS_TICK_CNT) / faktor;
	ELSE
		IF mode THEN
		    T_PLC_MS := DINT_TO_UDINT(PLC_SYS_TICK_CNT) / faktor;
		ELSE
		    T_PLC_MS := DINT_TO_UDINT(PLC_SYS_TICK_CNT) * faktor;
		END_IF;
	END_IF;

	IF debug THEN
		T_PLC_MS := (DWORD_TO_UDINT(SHL(UDINT_TO_DWORD(T_PLC_MS),N) OR SHL(temp,N)) - UDINT#1) + Offset;
	END_IF;

END_FUNCTION_BLOCK

FUNCTION TIME_TO_REAL1:REAL

	VAR_INPUT
		X :	TIME;
	END_VAR

	TIME_TO_REAL1 := UDINT_TO_REAL(DINT_TO_UDINT(TIME_TO_DINT(X)));
END_FUNCTION

FUNCTION MODR : REAL
  VAR_INPUT
    IN : REAL;
    DIVI : REAL;
  END_VAR

  IF divi = 0.0 THEN
  	MODR := 0.0;
  ELSE
  	MODR := in - DINT_TO_REAL(FLOOR2(in / divi)) * divi;
  END_IF;
END_FUNCTION

FUNCTION FLOOR2 : DINT
  VAR_INPUT
    x : REAL;
  END_VAR

  FLOOR2 := REAL_TO_DINT(X);
  IF DINT_TO_REAL(FLOOR2) > X THEN
  	FLOOR2 := FLOOR2 - DINT#1;
  END_IF;
END_FUNCTION

FUNCTION SIGN_R : BOOL
  VAR_INPUT
    IN : REAL;
  END_VAR

  SIGN_R := in < 0.0;
END_FUNCTION

FUNCTION_BLOCK GEN_SIN_Block

	VAR_INPUT
		PT :	TIME;
		AM :	REAL := REAL#1.0;
		OS :	REAL;
		DL :	REAL;
	END_VAR

	VAR_OUTPUT
		Q :	BOOL;
		Out :	REAL;
	END_VAR

	VAR
		tx :	TIME;
		last :	TIME;
		init :	BOOL;
		temp :	REAL;
		T_PLC_MS :	T_PLC_MS_Block;
	END_VAR

	T_PLC_MS();
	tx:= UDINT_TO_TIME(T_PLC_MS.T_PLC_MS) - last;

	DL := modR(dl,1.0);
	IF dl < 0.0 THEN dl := 1.0 - dl; END_IF;

	IF NOT init THEN
		init := TRUE;
		last := tx;
		tx := t#0s;
	END_IF;

	IF tx >= pt THEN
		last := last + pt;
		tx := tx - pt;
	END_IF;

	IF pt > t#0s THEN temp := SIN(6.283185307179586476 * TIME_TO_REAL1(tx + multime(pt, dl)) / TIME_TO_REAL(pt)); END_IF;
	out := am * 0.5 *  temp + os;

	q := NOT sign_R(temp);

END_FUNCTION_BLOCK

PROGRAM program0
  VAR
	PT :	TIME := T#1s;
	AM :	REAL := REAL#1.0;
	OS :	REAL;
	DL :	REAL;
	Q :	BOOL;
	OUT :	REAL;
	func_block : GEN_SIN_Block;
  END_VAR
	func_block.PT  :=PT;
	func_block.AM  :=AM;
	func_block.OS  :=OS;
	func_block.DL  :=DL;
	func_block();
	Q := func_block.Q;
	OUT := func_block.OUT;
END_PROGRAM

CONFIGURATION Config0
	VAR_GLOBAL
		PLC_TICKS_PER_SEC :	INT;
		PLC_SYS_TICK_CNT :	DINT;
	END_VAR
	RESOURCE Res0 ON PLC
		TASK task0(INTERVAL := T#20ms,PRIORITY := 0);
		PROGRAM instance0 WITH task0 : program0;
	END_RESOURCE
END_CONFIGURATION
